  MoveL 3421 to (458.38, 544.47, 60) mm, rotated rx 180 ry 0 rz 160 deg; joints [12.908, 64.671, 4.194, -145.247, 72.379, 168.139]
  Call Extruder(250.39892)
  MoveL 3422 to (457.49, 543.62, 60) mm, rotated rx -180 ry 0 rz 160 deg; joints [12.822, 64.543, 4.5, -145.367, 72.508, 168.272]
  Call Extruder(254.47184)
  MoveL 3423 to (456.59, 542.72, 60) mm, rotated rx -180 ry 0 rz 160 deg; joints [12.729, 64.414, 4.81, -145.496, 72.639, 168.409]
  Set speed (17.7 mm/s)
  Call Extruder(258.50937)
  MoveL 3424 to (455.71, 541.81, 60) mm, rotated rx -180 ry 0 rz 160 deg; joints [12.633, 64.289, 5.114, -145.625, 72.766, 168.543]
  Call Extruder(262.39777)
  MoveL 3425 to (454.88, 540.92, 60) mm, rotated rx 180 ry 0 rz 160 deg; joints [12.537, 64.17, 5.4, -145.753, 72.886, 168.671]
  Set speed (17.7 mm/s)
  Call Extruder(266.46406)
  MoveL 3426 to (454.04, 539.97, 60) mm, rotated rx -180 ry 0 rz 160 deg; joints [12.434, 64.049, 5.695, -145.888, 73.009, 168.804]
  Set speed (17.7 mm/s)
  Call Extruder(270.34791)
  MoveL 3427 to (453.25, 539.04, 60) mm, rotated rx -180 ry 0 rz 160 deg; joints [12.332, 63.935, 5.97, -146.021, 73.124, 168.929]
  Call Extruder(274.31271)
  MoveL 3428 to (452.46, 538.08, 60) mm, rotated rx 180 ry 0 rz 160 deg; joints [12.225, 63.822, 6.246, -146.158, 73.238, 169.056]
  Set speed (17.7 mm/s)
  Call Extruder(278.33345)
  MoveL 3429 to (451.68, 537.1, 60) mm, rotated rx 180 ry 0 rz 160 deg; joints [12.113, 63.71, 6.52, -146.3, 73.352, 169.183]
  Call Extruder(282.32372)
  MoveL 3430 to (450.94, 536.1, 60) mm, rotated rx 180 ry 0 rz 160 deg; joints [11.998, 63.601, 6.786, -146.444, 73.461, 169.307]
  Set speed (17.7 mm/s)
  Call Extruder(286.28959)
  MoveL 3431 to (450.21, 535.09, 60) mm, rotated rx 180 ry 0 rz 160 deg; joints [11.88, 63.495, 7.044, -146.589, 73.567, 169.429]
  Call Extruder(290.26148)
  MoveL 3432 to (449.5, 534.06, 60) mm, rotated rx -180 ry 0 rz 160 deg; joints [11.76, 63.392, 7.297, -146.736, 73.67, 169.55]
  Call Extruder(294.32502)
  MoveL 3433 to (448.81, 533, 60) mm, rotated rx 180 ry 0 rz 160 deg; joints [11.634, 63.29, 7.549, -146.89, 73.772, 169.671]
  Set speed (17.7 mm/s)
  Call Extruder(298.26201)
  MoveL 3434 to (448.15, 531.96, 60) mm, rotated rx 180 ry 0 rz 160 deg; joints [11.508, 63.193, 7.787, -147.041, 73.868, 169.787]
  Set speed (17.7 mm/s)
  Call Extruder(302.15383)
  MoveL 3435 to (447.52, 530.92, 60) mm, rotated rx -180 ry 0 rz 160 deg; joints [11.381, 63.1, 8.016, -147.192, 73.96, 169.9]
  Set speed (17.6 mm/s)
  Call Extruder(306.26935)
  MoveL 3436 to (446.88, 529.8, 60) mm, rotated rx 180 ry 0 rz 160 deg; joints [11.244, 63.005, 8.252, -147.355, 74.054, 170.018]
  Set speed (17.6 mm/s)
  Call Extruder(310.11261)
  MoveL 3437 to (446.3, 528.75, 60) mm, rotated rx 180 ry 0 rz 160 deg; joints [11.113, 62.918, 8.466, -147.508, 74.139, 170.126]
  Set speed (17.7 mm/s)
  Call Extruder(314.10849)
  MoveL 3438 to (445.72, 527.64, 60) mm, rotated rx 180 ry 0 rz 160 deg; joints [10.974, 62.831, 8.682, -147.67, 74.224, 170.237]
  Set speed (17.7 mm/s)
  Call Extruder(318.14964)
  MoveL 3439 to (445.16, 526.51, 60) mm, rotated rx 180 ry 0 rz 160 deg; joints [10.831, 62.746, 8.893, -147.836, 74.307, 170.347]
  Set speed (17.7 mm/s)
  Call Extruder(325.99805)
  MoveL 3440 to (444.13, 524.27, 60) mm, rotated rx 180 ry 0 rz 160 deg; joints [10.544, 62.589, 9.284, -148.164, 74.457, 170.554]
  Set speed (17.6 mm/s)
  Call Extruder(330.16567)
  MoveL 3441 to (443.63, 523.07, 60) mm, rotated rx -180 ry 0 rz 160 deg; joints [10.388, 62.511, 9.478, -148.341, 74.531, 170.661]
  Call Extruder(334.15174)
  MoveL 3442 to (443.17, 521.91, 60) mm, rotated rx -180 ry 0 rz 160 deg; joints [10.236, 62.438, 9.66, -148.512, 74.6, 170.761]
  Set speed (17.7 mm/s)
  Call Extruder(342.11094)
  MoveL 3443 to (442.32, 519.57, 60) mm, rotated rx 180 ry 0 rz 160 deg; joints [9.926, 62.302, 10.001, -148.858, 74.725, 170.955]
  Set speed (17.6 mm/s)
  Call Extruder(346.07808)
  MoveL 3444 to (441.94, 518.39, 60) mm, rotated rx 180 ry 0 rz 160 deg; joints [9.768, 62.24, 10.157, -149.034, 74.781, 171.048]
  Set speed (17.6 mm/s)
  Call Extruder(350.09490)
  MoveL 3445 to (441.57, 517.19, 60) mm, rotated rx 180 ry 0 rz 160 deg; joints [9.606, 62.179, 10.312, -149.212, 74.836, 171.141]
  Set speed (17.6 mm/s)
  Call Extruder(354.07902)
  MoveL 3446 to (441.23, 516, 60) mm, rotated rx -180 ry 0 rz 160 deg; joints [9.443, 62.122, 10.456, -149.391, 74.885, 171.231]
  Set speed (17.6 mm/s)
  Call Extruder(357.89675)
  MoveL 3447 to (440.93, 514.84, 60) mm, rotated rx 180 ry 0 rz 160 deg; joints [9.286, 62.069, 10.589, -149.563, 74.931, 171.315]
  Set speed (17.6 mm/s)
  Call Extruder(362.02810)
  MoveL 3448 to (440.63, 513.59, 60) mm, rotated rx -180 ry 0 rz 160 deg; joints [9.113, 62.016, 10.722, -149.751, 74.974, 171.403]
  Set speed (17.6 mm/s)
  Call Extruder(366.00274)
  MoveL 3449 to (440.36, 512.37, 60) mm, rotated rx -180 ry 0 rz 160 deg; joints [8.945, 61.967, 10.845, -149.933, 75.014, 171.486]
  Set speed (17.7 mm/s)
  Call Extruder(374.01194)
  MoveL 3450 to (439.9, 509.91, 60) mm, rotated rx 180 ry 0 rz 160 deg; joints [8.601, 61.878, 11.069, -150.303, 75.081, 171.647]
  Set speed (17.7 mm/s)
  Call Extruder(381.96597)
  MoveL 3451 to (439.55, 507.44, 60) mm, rotated rx 180 ry 0 rz 160 deg; joints [8.253, 61.803, 11.261, -150.674, 75.131, 171.797]
  Set speed (17.7 mm/s)
  Call Extruder(389.93168)
  MoveL 3452 to (439.29, 504.96, 60) mm, rotated rx 180 ry 0 rz 160 deg; joints [7.9, 61.739, 11.422, -151.049, 75.167, 171.939]
  Set speed (17.7 mm/s)
  Call Extruder(397.72230)
  MoveL 3453 to (439.14, 502.53, 60) mm, rotated rx -180 ry 0 rz 160 deg; joints [7.551, 61.689, 11.55, -151.416, 75.186, 172.069]
  Set speed (17.7 mm/s)
  Call Extruder(405.77297)
  MoveL 3454 to (439.09, 500.01, 60) mm, rotated rx 180 ry 0 rz 160 deg; joints [7.186, 61.649, 11.651, -151.798, 75.19, 172.195]
  Set speed (17.7 mm/s)
  Call Extruder(413.01680)
  MoveL 3455 to (439.13, 497.74, 60) mm, rotated rx 180 ry 0 rz 160 deg; joints [6.856, 61.624, 11.714, -152.141, 75.179, 172.3]
  Set speed (17.7 mm/s)
  Call Extruder(420.09250)
  MoveL 3456 to (439.25, 495.53, 60) mm, rotated rx 180 ry 0 rz 160 deg; joints [6.532, 61.61, 11.75, -152.476, 75.156, 172.396]
  Set speed (17.7 mm/s)
  Call Extruder(427.18898)
  MoveL 3457 to (439.46, 493.32, 60) mm, rotated rx 180 ry 0 rz 160 deg; joints [6.207, 61.606, 11.762, -152.81, 75.119, 172.485]
  Set speed (17.7 mm/s)
  Call Extruder(434.08176)
  MoveL 3458 to (439.73, 491.18, 60) mm, rotated rx 180 ry 0 rz 160 deg; joints [5.891, 61.611, 11.749, -153.133, 75.071, 172.564]
  Call Extruder(441.67457)
  MoveL 3459 to (440.12, 488.84, 60) mm, rotated rx -180 ry 0 rz 160 deg; joints [5.544, 61.627, 11.708, -153.487, 75.004, 172.645]
  Set speed (17.7 mm/s)
  Call Extruder(448.69639)
  MoveL 3460 to (440.56, 486.69, 60) mm, rotated rx 180 ry 0 rz 160 deg; joints [5.224, 61.652, 11.644, -153.811, 74.929, 172.712]
  Call Extruder(455.92149)
  MoveL 3461 to (441.1, 484.49, 60) mm, rotated rx 180 ry 0 rz 160 deg; joints [4.897, 61.687, 11.554, -154.14, 74.838, 172.775]
  Call Extruder(462.99323)
  MoveL 3462 to (441.7, 482.36, 60) mm, rotated rx 180 ry 0 rz 160 deg; joints [4.579, 61.732, 11.44, -154.459, 74.736, 172.83]
  Set speed (17.7 mm/s)
  Call Extruder(470.18160)
  MoveL 3463 to (442.39, 480.22, 60) mm, rotated rx -180 ry 0 rz 160 deg; joints [4.26, 61.788, 11.299, -154.777, 74.619, 172.878]
  Set speed (17.7 mm/s)
  Call Extruder(477.50769)
  MoveL 3464 to (443.18, 478.07, 60) mm, rotated rx 180 ry 0 rz 160 deg; joints [3.939, 61.855, 11.129, -155.096, 74.486, 172.921]
  Set speed (17.7 mm/s)
  Call Extruder(484.67427)
  MoveL 3465 to (444.02, 475.99, 60) mm, rotated rx 180 ry 0 rz 160 deg; joints [3.629, 61.93, 10.939, -155.401, 74.344, 172.957]
  Set speed (17.7 mm/s)
  Call Extruder(491.67065)
  MoveL 3466 to (444.92, 473.99, 60) mm, rotated rx -180 ry 0 rz 160 deg; joints [3.332, 62.013, 10.729, -155.693, 74.192, 172.986]
  Set speed (17.7 mm/s)
  Call Extruder(499.01562)
  MoveL 3467 to (445.94, 471.93, 60) mm, rotated rx -180 ry 0 rz 160 deg; joints [3.026, 62.111, 10.483, -155.992, 74.019, 173.009]
  Set speed (17.6 mm/s)
  Call Extruder(506.01239)
  MoveL 3468 to (446.99, 470.01, 60) mm, rotated rx 180 ry 0 rz 160 deg; joints [2.74, 62.212, 10.227, -156.269, 73.844, 173.026]
  Set speed (17.7 mm/s)
  Call Extruder(513.18194)
  MoveL 3469 to (448.13, 468.08, 60) mm, rotated rx -180 ry 0 rz 160 deg; joints [2.455, 62.326, 9.941, -156.544, 73.651, 173.037]
  Set speed (17.7 mm/s)
  Call Extruder(520.42302)
  MoveL 3470 to (449.35, 466.17, 60) mm, rotated rx -180 ry 0 rz 160 deg; joints [2.173, 62.451, 9.628, -156.813, 73.445, 173.042]
  Set speed (17.7 mm/s)
  Call Extruder(527.57955)
  MoveL 3471 to (450.62, 464.33, 60) mm, rotated rx -180 ry 0 rz 160 deg; joints [1.903, 62.584, 9.296, -157.07, 73.229, 173.041]
  Set speed (17.7 mm/s)
  Call Extruder(534.77776)
  MoveL 3472 to (451.98, 462.53, 60) mm, rotated rx -180 ry 0 rz 160 deg; joints [1.64, 62.727, 8.94, -157.318, 73, 173.033]
  Call Extruder(541.94995)
  MoveL 3473 to (453.39, 460.79, 60) mm, rotated rx 180 ry 0 rz 160 deg; joints [1.386, 62.88, 8.562, -157.555, 72.761, 173.02]
  Set speed (17.7 mm/s)
  Call Extruder(549.06578)
  MoveL 3474 to (454.86, 459.11, 60) mm, rotated rx 180 ry 0 rz 160 deg; joints [1.143, 63.039, 8.166, -157.779, 72.513, 173.002]
  Set speed (17.7 mm/s)
  Call Extruder(556.16490)
  MoveL 3475 to (456.38, 457.49, 60) mm, rotated rx 180 ry 0 rz 160 deg; joints [0.91, 63.208, 7.75, -157.993, 72.256, 172.978]
  Set speed (17.7 mm/s)
  Call Extruder(563.37874)
  MoveL 3476 to (457.99, 455.9, 60) mm, rotated rx -180 ry 0 rz 160 deg; joints [0.683, 63.388, 7.308, -158.198, 71.984, 172.947]
  Set speed (17.7 mm/s)
  Call Extruder(570.70409)
  MoveL 3477 to (459.68, 454.35, 60) mm, rotated rx 180 ry 0 rz 160 deg; joints [0.463, 63.58, 6.837, -158.394, 71.698, 172.91]
  Set speed (17.7 mm/s)
  Call Extruder(577.80064)
  MoveL 3478 to (461.37, 452.91, 60) mm, rotated rx 180 ry 0 rz 160 deg; joints [0.26, 63.774, 6.362, -158.571, 71.412, 172.869]
  Set speed (17.7 mm/s)
  Call Extruder(584.88132)
  MoveL 3479 to (463.11, 451.53, 60) mm, rotated rx 180 ry 0 rz 160 deg; joints [0.068, 63.977, 5.87, -158.737, 71.118, 172.822]
  Set speed (17.7 mm/s)
  Call Extruder(592.12824)
  MoveL 3480 to (464.94, 450.19, 60) mm, rotated rx -180 ry 0 rz 160 deg; joints [-0.118, 64.192, 5.348, -158.893, 70.809, 172.769]
  Set speed (17.7 mm/s)
  Call Extruder(599.20393)
  MoveL 3481 to (466.77, 448.95, 60) mm, rotated rx -180 ry 0 rz 160 deg; joints [-0.288, 64.41, 4.82, -159.034, 70.499, 172.71]
  Set speed (17.7 mm/s)
  Call Extruder(606.45847)
  MoveL 3482 to (468.7, 447.75, 60) mm, rotated rx 180 ry 0 rz 160 deg; joints [-0.452, 64.642, 4.262, -159.164, 70.173, 172.645]
  Set speed (17.7 mm/s)
  Call Extruder(613.61813)
  MoveL 3483 to (470.64, 446.63, 60) mm, rotated rx 180 ry 0 rz 160 deg; joints [-0.602, 64.879, 3.695, -159.28, 69.845, 172.574]
  Set speed (17.7 mm/s)
  Call Extruder(620.78178)
  MoveL 3484 to (472.62, 445.59, 60) mm, rotated rx 180 ry 0 rz 160 deg; joints [-0.741, 65.123, 3.112, -159.383, 69.509, 172.498]
  Set speed (17.7 mm/s)
  Call Extruder(627.85751)
  MoveL 3485 to (474.62, 444.63, 60) mm, rotated rx -180 ry 0 rz 160 deg; joints [-0.867, 65.372, 2.52, -159.471, 69.172, 172.416]
  Call Extruder(635.11103)
  MoveL 3486 to (476.7, 443.72, 60) mm, rotated rx -180 ry 0 rz 160 deg; joints [-0.985, 65.633, 1.9, -159.548, 68.82, 172.326]
  Set speed (17.7 mm/s)
  Call Extruder(642.12717)
  MoveL 3487 to (478.75, 442.92, 60) mm, rotated rx -180 ry 0 rz 160 deg; joints [-1.087, 65.894, 1.286, -159.609, 68.475, 172.233]
  Set speed (17.7 mm/s)
  Call Extruder(649.44940)
  MoveL 3488 to (480.91, 442.16, 60) mm, rotated rx 180 ry 0 rz 160 deg; joints [-1.183, 66.172, 0.632, -159.659, 68.109, 172.13]
  Set speed (17.7 mm/s)
  Call Extruder(656.54664)
  MoveL 3489 to (483.03, 441.5, 60) mm, rotated rx 180 ry 0 rz 160 deg; joints [-1.264, 66.447, -0.015, -159.694, 67.751, 172.024]
  Set speed (17.7 mm/s)
  Call Extruder(663.55363)
  MoveL 3490 to (485.15, 440.93, 60) mm, rotated rx -180 ry 0 rz 160 deg; joints [-1.334, 66.726, -0.664, -159.715, 67.393, 171.913]
  Call Extruder(670.92630)
  MoveL 3491 to (487.39, 440.41, 60) mm, rotated rx -180 ry 0 rz 160 deg; joints [-1.395, 67.024, -1.359, -159.723, 67.013, 171.79]
  Set speed (17.7 mm/s)
  Call Extruder(677.95259)
  MoveL 3492 to (489.55, 439.99, 60) mm, rotated rx -180 ry 0 rz 160 deg; joints [-1.442, 67.315, -2.031, -159.717, 66.647, 171.666]
  Call Extruder(684.84672)
  MoveL 3493 to (491.69, 439.66, 60) mm, rotated rx 180 ry 0 rz 160 deg; joints [-1.479, 67.604, -2.699, -159.699, 66.287, 171.538]
  Call Extruder(692.33816)
  MoveL 3494 to (494.01, 439.38, 60) mm, rotated rx -180 ry 0 rz 160 deg; joints [-1.506, 67.924, -3.435, -159.665, 65.893, 171.392]
  Set speed (17.7 mm/s)
  Call Extruder(699.51358)
  MoveL 3495 to (496.25, 439.21, 60) mm, rotated rx 180 ry 0 rz 160 deg; joints [-1.522, 68.236, -4.148, -159.619, 65.514, 171.246]
  Call Extruder(706.76277)
  MoveL 3496 to (498.52, 439.11, 60) mm, rotated rx 180 ry 0 rz 160 deg; joints [-1.527, 68.554, -4.876, -159.559, 65.13, 171.091]
  Call Extruder(713.85821)
  MoveL 3497 to (500.74, 439.1, 60) mm, rotated rx -180 ry 0 rz 160 deg; joints [-1.521, 68.871, -5.595, -159.486, 64.754, 170.933]
  Set speed (17.7 mm/s)
  Call Extruder(720.88825)
  MoveL 3498 to (502.94, 439.16, 60) mm, rotated rx 180 ry 0 rz 160 deg; joints [-1.505, 69.187, -6.313, -159.402, 64.381, 170.77]
  Call Extruder(728.18043)
  MoveL 3499 to (505.22, 439.31, 60) mm, rotated rx 180 ry 0 rz 160 deg; joints [-1.478, 69.52, -7.063, -159.301, 63.994, 170.593]
  Set speed (17.7 mm/s)
  Call Extruder(735.41102)
  MoveL 3500 to (507.47, 439.55, 60) mm, rotated rx 180 ry 0 rz 160 deg; joints [-1.441, 69.852, -7.81, -159.188, 63.612, 170.411]
  Set speed (17.7 mm/s)
  Call Extruder(742.49479)
  MoveL 3501 to (509.66, 439.86, 60) mm, rotated rx 180 ry 0 rz 160 deg; joints [-1.396, 70.18, -8.545, -159.065, 63.239, 170.227]
  Set speed (17.6 mm/s)
  Call Extruder(749.70308)
  MoveL 3502 to (511.88, 440.26, 60) mm, rotated rx -180 ry 0 rz 160 deg; joints [-1.339, 70.515, -9.296, -158.928, 62.862, 170.032]
  Set speed (17.7 mm/s)
  Call Extruder(756.88945)
  MoveL 3503 to (514.08, 440.74, 60) mm, rotated rx -180 ry 0 rz 160 deg; joints [-1.274, 70.852, -10.045, -158.778, 62.488, 169.83]
  Set speed (17.7 mm/s)
  Call Extruder(763.93252)
  MoveL 3504 to (516.21, 441.29, 60) mm, rotated rx 180 ry 0 rz 160 deg; joints [-1.201, 71.183, -10.781, -158.619, 62.124, 169.627]
  Set speed (17.7 mm/s)
  Call Extruder(771.15493)
  MoveL 3505 to (518.38, 441.93, 60) mm, rotated rx 180 ry 0 rz 160 deg; joints [-1.116, 71.524, -11.536, -158.445, 61.754, 169.411]
  Call Extruder(778.20140)
  MoveL 3506 to (520.47, 442.63, 60) mm, rotated rx -180 ry 0 rz 160 deg; joints [-1.026, 71.857, -12.271, -158.263, 61.398, 169.194]
  Set speed (17.7 mm/s)
  Call Extruder(785.48617)
  MoveL 3507 to (522.61, 443.44, 60) mm, rotated rx -180 ry 0 rz 160 deg; joints [-0.923, 72.202, -13.029, -158.064, 61.033, 168.964]
  Set speed (17.7 mm/s)
  Call Extruder(792.88462)
  MoveL 3508 to (524.74, 444.34, 60) mm, rotated rx 180 ry 0 rz 160 deg; joints [-0.81, 72.551, -13.795, -157.85, 60.669, 168.722]
  Set speed (17.7 mm/s)
  Call Extruder(799.85949)
  MoveL 3509 to (526.72, 445.26, 60) mm, rotated rx 180 ry 0 rz 160 deg; joints [-0.696, 72.88, -14.515, -157.637, 60.33, 168.489]
  Set speed (17.7 mm/s)
  Call Extruder(807.02755)
  MoveL 3510 to (528.71, 446.28, 60) mm, rotated rx 180 ry 0 rz 160 deg; joints [-0.57, 73.217, -15.249, -157.409, 59.988, 168.244]
  Set speed (17.7 mm/s)
  Call Extruder(814.23835)
  MoveL 3511 to (530.68, 447.38, 60) mm, rotated rx 180 ry 0 rz 160 deg; joints [-0.437, 73.554, -15.981, -157.169, 59.65, 167.991]
  Set speed (17.7 mm/s)
  Call Extruder(821.30859)
  MoveL 3512 to (532.58, 448.53, 60) mm, rotated rx -180 ry 0 rz 160 deg; joints [-0.299, 73.882, -16.693, -156.924, 59.326, 167.738]
  Call Extruder(828.55700)
  MoveL 3513 to (534.47, 449.78, 60) mm, rotated rx -180 ry 0 rz 160 deg; joints [-0.149, 74.215, -17.414, -156.663, 59.002, 167.473]
  Call Extruder(835.64231)
  MoveL 3514 to (536.27, 451.07, 60) mm, rotated rx 180 ry 0 rz 160 deg; joints [0.003, 74.538, -18.111, -156.399, 58.693, 167.209]
  Set speed (17.7 mm/s)
  Call Extruder(842.84270)
  MoveL 3515 to (538.06, 452.45, 60) mm, rotated rx 180 ry 0 rz 160 deg; joints [0.165, 74.863, -18.81, -156.122, 58.386, 166.936]
  Set speed (17.7 mm/s)
  Call Extruder(850.00063)
  MoveL 3516 to (539.78, 453.88, 60) mm, rotated rx 180 ry 0 rz 160 deg; joints [0.332, 75.181, -19.492, -155.838, 58.091, 166.66]
  Set speed (17.7 mm/s)
  Call Extruder(857.35471)
  MoveL 3517 to (541.5, 455.41, 60) mm, rotated rx -180 ry 0 rz 160 deg; joints [0.51, 75.503, -20.181, -155.539, 57.798, 166.373]
  Set speed (17.7 mm/s)
  Call Extruder(864.32574)
  MoveL 3518 to (543.07, 456.93, 60) mm, rotated rx -180 ry 0 rz 160 deg; joints [0.685, 75.803, -20.823, -155.249, 57.529, 166.098]
  Set speed (17.7 mm/s)
  Call Extruder(868.29280)
  MoveL 3519 to (543.94, 457.82, 60) mm, rotated rx -180 ry 0 rz 160 deg; joints [0.787, 75.97, -21.18, -155.08, 57.382, 165.94]
  Set speed (17.7 mm/s)
  Call Extruder(872.16707)
  MoveL 3520 to (544.77, 458.7, 60) mm, rotated rx 180 ry 0 rz 160 deg; joints [0.888, 76.133, -21.526, -154.914, 57.24, 165.785]
  Set speed (17.7 mm/s)
  Call Extruder(876.17456)
  MoveL 3521 to (545.61, 459.63, 60) mm, rotated rx -180 ry 0 rz 160 deg; joints [0.994, 76.298, -21.879, -154.74, 57.097, 165.624]
  Call Extruder(880.12274)
  MoveL 3522 to (546.42, 460.56, 60) mm, rotated rx -180 ry 0 rz 160 deg; joints [1.1, 76.46, -22.222, -154.567, 56.959, 165.464]
  Set speed (17.7 mm/s)
  Call Extruder(884.11982)
  MoveL 3523 to (547.22, 461.52, 60) mm, rotated rx -180 ry 0 rz 160 deg; joints [1.209, 76.621, -22.564, -154.39, 56.823, 165.302]
  Set speed (17.7 mm/s)
  Call Extruder(888.15091)
  MoveL 3524 to (548.01, 462.51, 60) mm, rotated rx 180 ry 0 rz 160 deg; joints [1.321, 76.78, -22.903, -154.21, 56.69, 165.139]
  Set speed (17.7 mm/s)
  Call Extruder(892.09605)
  MoveL 3525 to (548.76, 463.49, 60) mm, rotated rx 180 ry 0 rz 160 deg; joints [1.432, 76.934, -23.228, -154.033, 56.564, 164.978]
  Set speed (17.7 mm/s)
  Call Extruder(896.05523)
  MoveL 3526 to (549.49, 464.49, 60) mm, rotated rx -180 ry 0 rz 160 deg; joints [1.545, 77.086, -23.55, -153.853, 56.441, 164.817]
  Call Extruder(900.07180)
  MoveL 3527 to (550.21, 465.52, 60) mm, rotated rx -180 ry 0 rz 160 deg; joints [1.66, 77.237, -23.87, -153.669, 56.32, 164.653]
  Set speed (17.6 mm/s)
  Call Extruder(904.02046)
  MoveL 3528 to (550.9, 466.55, 60) mm, rotated rx -180 ry 0 rz 160 deg; joints [1.775, 77.383, -24.179, -153.488, 56.205, 164.492]
  Set speed (17.7 mm/s)
  Call Extruder(908.03453)
  MoveL 3529 to (551.58, 467.6, 60) mm, rotated rx 180 ry 0 rz 160 deg; joints [1.894, 77.529, -24.487, -153.302, 56.092, 164.328]
  Call Extruder(912.01280)
  MoveL 3530 to (552.23, 468.66, 60) mm, rotated rx -180 ry 0 rz 160 deg; joints [2.012, 77.67, -24.785, -153.116, 55.984, 164.166]
  Set speed (17.7 mm/s)
  Call Extruder(916.05485)
  MoveL 3531 to (552.87, 469.75, 60) mm, rotated rx 180 ry 0 rz 160 deg; joints [2.134, 77.811, -25.081, -152.927, 55.879, 164.002]
  Set speed (17.6 mm/s)
  Call Extruder(921.15306)
  MoveL 3532 to (553.65, 471.15, 60) mm, rotated rx -180 ry 0 rz 160 deg; joints [2.289, 77.983, -25.444, -152.688, 55.753, 163.795]
  Call Extruder(923.98862)
  MoveL 3533 to (554.06, 471.93, 60) mm, rotated rx 180 ry 0 rz 160 deg; joints [2.376, 78.076, -25.639, -152.554, 55.686, 163.681]
  Set speed (17.7 mm/s)
  Call Extruder(927.92565)
  MoveL 3534 to (554.61, 473.03, 60) mm, rotated rx 180 ry 0 rz 160 deg; joints [2.498, 78.204, -25.907, -152.368, 55.596, 163.523]
  Set speed (17.7 mm/s)
  Call Extruder(931.94237)
  MoveL 3535 to (555.16, 474.16, 60) mm, rotated rx 180 ry 0 rz 160 deg; joints [2.624, 78.33, -26.171, -152.178, 55.509, 163.362]
  Set speed (17.7 mm/s)
  Call Extruder(935.87944)
  MoveL 3536 to (555.67, 475.28, 60) mm, rotated rx -180 ry 0 rz 160 deg; joints [2.748, 78.45, -26.424, -151.991, 55.428, 163.205]
  Set speed (17.6 mm/s)
  Call Extruder(943.97320)
  MoveL 3537 to (556.65, 477.62, 60) mm, rotated rx -180 ry 0 rz 160 deg; joints [3.007, 78.685, -26.916, -151.606, 55.277, 162.886]
  Set speed (17.6 mm/s)
  Call Extruder(947.91335)
  MoveL 3538 to (557.08, 478.77, 60) mm, rotated rx 180 ry 0 rz 160 deg; joints [3.134, 78.792, -27.141, -151.419, 55.211, 162.733]
  Set speed (17.6 mm/s)
  Call Extruder(951.77830)
  MoveL 3539 to (557.5, 479.9, 60) mm, rotated rx -180 ry 0 rz 160 deg; joints [3.259, 78.896, -27.358, -151.236, 55.149, 162.584]
  Call Extruder(955.89683)
  MoveL 3540 to (557.91, 481.12, 60) mm, rotated rx -180 ry 0 rz 160 deg; joints [3.394, 79.001, -27.577, -151.041, 55.09, 162.427]
  Set speed (17.6 mm/s)
  Call Extruder(959.91891)
  MoveL 3541 to (558.29, 482.32, 60) mm, rotated rx 180 ry 0 rz 160 deg; joints [3.526, 79.101, -27.786, -150.85, 55.034, 162.275]
  Set speed (17.7 mm/s)
  Call Extruder(967.71701)
  MoveL 3542 to (558.95, 484.67, 60) mm, rotated rx 180 ry 0 rz 160 deg; joints [3.785, 79.28, -28.16, -150.482, 54.944, 161.985]
  Set speed (17.6 mm/s)
  Call Extruder(971.84165)
  MoveL 3543 to (559.26, 485.92, 60) mm, rotated rx -180 ry 0 rz 160 deg; joints [3.924, 79.366, -28.34, -150.289, 54.905, 161.836]
  Call Extruder(975.71381)
  MoveL 3544 to (559.53, 487.1, 60) mm, rotated rx 180 ry 0 rz 160 deg; joints [4.054, 79.446, -28.506, -150.108, 54.871, 161.697]
  Set speed (17.7 mm/s)
  Call Extruder(983.59562)
  MoveL 3545 to (560, 489.52, 60) mm, rotated rx 180 ry 0 rz 160 deg; joints [4.321, 79.591, -28.808, -149.742, 54.82, 161.422]
  Set speed (17.7 mm/s)
  Call Extruder(991.63549)
  MoveL 3546 to (560.38, 492.01, 60) mm, rotated rx -180 ry 0 rz 160 deg; joints [4.596, 79.721, -29.079, -149.374, 54.787, 161.152]
  Set speed (17.7 mm/s)
  Call Extruder(999.76645)
  MoveL 3547 to (560.67, 494.54, 60) mm, rotated rx -180 ry 0 rz 160 deg; joints [4.875, 79.832, -29.31, -149.006, 54.774, 160.889]
  Call Extruder(1007.63307)
  MoveL 3548 to (560.84, 497, 60) mm, rotated rx -180 ry 0 rz 160 deg; joints [5.148, 79.92, -29.493, -148.657, 54.783, 160.648]
  Set speed (17.7 mm/s)
  Call Extruder(1015.58635)
  MoveL 3549 to (560.91, 499.49, 60) mm, rotated rx -180 ry 0 rz 160 deg; joints [5.424, 79.989, -29.637, -148.311, 54.811, 160.416]
  Set speed (17.7 mm/s)
  Call Extruder(1023.42990)
  MoveL 3550 to (560.88, 501.94, 60) mm, rotated rx 180 ry 0 rz 160 deg; joints [5.698, 80.037, -29.736, -147.977, 54.859, 160.201]
  Set speed (17.7 mm/s)
  Call Extruder(1031.49963)
  MoveL 3551 to (560.75, 504.46, 60) mm, rotated rx 180 ry 0 rz 160 deg; joints [5.98, 80.066, -29.796, -147.641, 54.929, 159.995]
  Call Extruder(1039.46843)
  MoveL 3552 to (560.51, 506.95, 60) mm, rotated rx 180 ry 0 rz 160 deg; joints [6.258, 80.073, -29.812, -147.318, 55.018, 159.806]
  Call Extruder(1047.51753)
  MoveL 3553 to (560.17, 509.45, 60) mm, rotated rx -180 ry 0 rz 160 deg; joints [6.54, 80.059, -29.783, -147.002, 55.128, 159.632]
  Set speed (17.7 mm/s)
  Call Extruder(1055.37383)
  MoveL 3554 to (559.74, 511.87, 60) mm, rotated rx 180 ry 0 rz 160 deg; joints [6.814, 80.026, -29.714, -146.702, 55.254, 159.477]
  Call Extruder(1063.39954)
  MoveL 3555 to (559.2, 514.32, 60) mm, rotated rx 180 ry 0 rz 160 deg; joints [7.094, 79.971, -29.6, -146.407, 55.402, 159.335]
  Set speed (17.7 mm/s)
  Call Extruder(1071.21656)
  MoveL 3556 to (558.58, 516.69, 60) mm, rotated rx -180 ry 0 rz 160 deg; joints [7.365, 79.898, -29.447, -146.129, 55.564, 159.214]
  Set speed (17.6 mm/s)
  Call Extruder(1075.37612)
  MoveL 3557 to (558.21, 517.93, 60) mm, rotated rx -180 ry 0 rz 160 deg; joints [7.508, 79.85, -29.347, -145.986, 55.658, 159.158]
  Set speed (17.6 mm/s)
  Call Extruder(1079.17724)
  MoveL 3558 to (557.85, 519.07, 60) mm, rotated rx -180 ry 0 rz 160 deg; joints [7.64, 79.804, -29.251, -145.857, 55.746, 159.108]
  Set speed (17.7 mm/s)
  Call Extruder(1087.36494)
  MoveL 3559 to (557, 521.48, 60) mm, rotated rx 180 ry 0 rz 160 deg; joints [7.921, 79.686, -29.006, -145.588, 55.951, 159.016]
  Set speed (17.7 mm/s)
  Call Extruder(1095.08205)
  MoveL 3560 to (556.1, 523.72, 60) mm, rotated rx 180 ry 0 rz 160 deg; joints [8.184, 79.556, -28.736, -145.346, 56.161, 158.947]
  Set speed (17.6 mm/s)
  Call Extruder(1099.19827)
  MoveL 3561 to (555.58, 524.9, 60) mm, rotated rx -180 ry 0 rz 160 deg; joints [8.323, 79.479, -28.575, -145.222, 56.28, 158.918]
  Set speed (17.6 mm/s)
  Call Extruder(1102.99136)
  MoveL 3562 to (555.09, 525.98, 60) mm, rotated rx 180 ry 0 rz 160 deg; joints [8.451, 79.405, -28.422, -145.108, 56.392, 158.893]
  Set speed (17.6 mm/s)
  Call Extruder(1105.96710)
  MoveL 3563 to (554.69, 526.82, 60) mm, rotated rx 180 ry 0 rz 160 deg; joints [8.551, 79.345, -28.296, -145.021, 56.482, 158.876]
  Set speed (17.6 mm/s)
  Call Extruder(1111.16558)
  MoveL 3564 to (553.96, 528.27, 60) mm, rotated rx -180 ry 0 rz 160 deg; joints [8.725, 79.232, -28.06, -144.874, 56.645, 158.854]
  Set speed (17.7 mm/s)
  Call Extruder(1115.08771)
  MoveL 3565 to (553.37, 529.35, 60) mm, rotated rx -180 ry 0 rz 160 deg; joints [8.855, 79.141, -27.87, -144.766, 56.772, 158.842]
  Set speed (17.6 mm/s)
  Call Extruder(1119.14376)
  MoveL 3566 to (552.75, 530.46, 60) mm, rotated rx 180 ry 0 rz 160 deg; joints [8.989, 79.043, -27.665, -144.657, 56.908, 158.834]
  Set speed (17.7 mm/s)
  Call Extruder(1122.98241)
  MoveL 3567 to (552.14, 531.49, 60) mm, rotated rx 180 ry 0 rz 160 deg; joints [9.115, 78.947, -27.464, -144.556, 57.039, 158.83]
  Set speed (17.7 mm/s)
  Call Extruder(1126.41961)
  MoveL 3568 to (551.57, 532.41, 60) mm, rotated rx 180 ry 0 rz 160 deg; joints [9.227, 78.857, -27.277, -144.469, 57.159, 158.83]
  Set speed (17.7 mm/s)
  Call Extruder(1131.07197)
  MoveL 3569 to (550.79, 533.63, 60) mm, rotated rx 180 ry 0 rz 160 deg; joints [9.378, 78.731, -27.013, -144.353, 57.326, 158.835]
  Set speed (17.7 mm/s)
  Call Extruder(1135.03970)
  MoveL 3570 to (550.09, 534.66, 60) mm, rotated rx -180 ry 0 rz 160 deg; joints [9.505, 78.619, -26.778, -144.258, 57.472, 158.844]
  Call Extruder(1138.93510)
  MoveL 3571 to (549.39, 535.65, 60) mm, rotated rx -180 ry 0 rz 160 deg; joints [9.63, 78.506, -26.54, -144.166, 57.617, 158.856]
  Call Extruder(1142.95939)
  MoveL 3572 to (548.64, 536.67, 60) mm, rotated rx 180 ry 0 rz 160 deg; joints [9.757, 78.385, -26.287, -144.075, 57.771, 158.873]
  Set speed (17.7 mm/s)
  Call Extruder(1146.90899)
  MoveL 3573 to (547.88, 537.65, 60) mm, rotated rx -180 ry 0 rz 160 deg; joints [9.881, 78.262, -26.03, -143.988, 57.925, 158.894]
  Set speed (17.7 mm/s)
  Call Extruder(1150.87614)
  MoveL 3574 to (547.11, 538.62, 60) mm, rotated rx 180 ry 0 rz 160 deg; joints [10.005, 78.136, -25.764, -143.903, 58.082, 158.918]
  Set speed (17.7 mm/s)
  Call Extruder(1154.87895)
  MoveL 3575 to (546.3, 539.57, 60) mm, rotated rx 180 ry 0 rz 160 deg; joints [10.129, 78.004, -25.488, -143.82, 58.243, 158.947]
  Set speed (17.7 mm/s)
  Call Extruder(1158.89048)
  MoveL 3576 to (545.48, 540.52, 60) mm, rotated rx 180 ry 0 rz 160 deg; joints [10.251, 77.87, -25.204, -143.74, 58.407, 158.98]
  Set speed (17.7 mm/s)
  Call Extruder(1162.94185)
  MoveL 3577 to (544.62, 541.46, 60) mm, rotated rx -180 ry 0 rz 160 deg; joints [10.374, 77.731, -24.911, -143.661, 58.575, 159.016]
  Set speed (17.6 mm/s)
  Call Extruder(1166.20153)
  MoveL 3578 to (543.92, 542.2, 60) mm, rotated rx -180 ry 0 rz 160 deg; joints [10.472, 77.616, -24.67, -143.6, 58.712, 159.049]
  Call Extruder(1170.78283)
  MoveL 3579 to (542.92, 543.22, 60) mm, rotated rx 180 ry 0 rz 160 deg; joints [10.607, 77.452, -24.324, -143.518, 58.907, 159.099]
  Set speed (17.7 mm/s)
  Call Extruder(1174.82308)
  MoveL 3580 to (542.01, 544.1, 60) mm, rotated rx -180 ry 0 rz 160 deg; joints [10.726, 77.304, -24.01, -143.448, 59.082, 159.147]
  Set speed (17.7 mm/s)
  Call Extruder(1178.74465)
  MoveL 3581 to (541.11, 544.94, 60) mm, rotated rx -180 ry 0 rz 160 deg; joints [10.839, 77.157, -23.7, -143.382, 59.253, 159.197]
  Call Extruder(1182.78523)
  MoveL 3582 to (540.17, 545.78, 60) mm, rotated rx 180 ry 0 rz 160 deg; joints [10.955, 77.003, -23.375, -143.317, 59.432, 159.252]
  Set speed (17.7 mm/s)
  Call Extruder(1186.72339)
  MoveL 3583 to (539.24, 546.59, 60) mm, rotated rx 180 ry 0 rz 160 deg; joints [11.066, 76.851, -23.052, -143.257, 59.608, 159.309]
  Set speed (17.7 mm/s)
  Call Extruder(1190.68443)
  MoveL 3584 to (538.28, 547.38, 60) mm, rotated rx -180 ry 0 rz 160 deg; joints [11.177, 76.695, -22.722, -143.198, 59.787, 159.369]
  Set speed (17.6 mm/s)
  Call Extruder(1194.72892)
  MoveL 3585 to (537.29, 548.16, 60) mm, rotated rx 180 ry 0 rz 160 deg; joints [11.288, 76.534, -22.379, -143.141, 59.971, 159.435]
  Set speed (17.6 mm/s)
  Call Extruder(1198.65969)
  MoveL 3586 to (536.31, 548.9, 60) mm, rotated rx 180 ry 0 rz 160 deg; joints [11.394, 76.374, -22.04, -143.088, 60.152, 159.502]
  Set speed (17.7 mm/s)
  Call Extruder(1202.66778)
  MoveL 3587 to (535.3, 549.64, 60) mm, rotated rx -180 ry 0 rz 160 deg; joints [11.501, 76.21, -21.69, -143.036, 60.338, 159.573]
  Set speed (17.7 mm/s)
  Call Extruder(1206.66997)
  MoveL 3588 to (534.27, 550.36, 60) mm, rotated rx -180 ry 0 rz 160 deg; joints [11.606, 76.043, -21.335, -142.987, 60.525, 159.647]
  Call Extruder(1210.71298)
  MoveL 3589 to (533.21, 551.06, 60) mm, rotated rx -180 ry 0 rz 160 deg; joints [11.711, 75.872, -20.971, -142.94, 60.715, 159.726]
  Set speed (17.7 mm/s)
  Call Extruder(1214.67331)
  MoveL 3590 to (532.17, 551.72, 60) mm, rotated rx 180 ry 0 rz 160 deg; joints [11.811, 75.704, -20.611, -142.896, 60.903, 159.805]
  Set speed (17.6 mm/s)
  Call Extruder(1218.61209)
  MoveL 3591 to (531.12, 552.36, 60) mm, rotated rx -180 ry 0 rz 160 deg; joints [11.91, 75.534, -20.248, -142.856, 61.091, 159.887]
  Set speed (17.6 mm/s)
  Call Extruder(1222.58771)
  MoveL 3592 to (530.04, 552.99, 60) mm, rotated rx -180 ry 0 rz 160 deg; joints [12.007, 75.361, -19.879, -142.817, 61.281, 159.973]
  Set speed (17.7 mm/s)
  Call Extruder(1226.49865)
  MoveL 3593 to (528.97, 553.58, 60) mm, rotated rx 180 ry 0 rz 160 deg; joints [12.101, 75.19, -19.511, -142.781, 61.469, 160.06]
  Set speed (17.7 mm/s)
  Call Extruder(1232.61058)
  MoveL 3594 to (527.27, 554.47, 60) mm, rotated rx 180 ry 0 rz 160 deg; joints [12.245, 74.918, -18.929, -142.729, 61.766, 160.2]
  Set speed (17.7 mm/s)
  Call Extruder(1238.37297)
  MoveL 3595 to (525.64, 555.25, 60) mm, rotated rx -180 ry 0 rz 160 deg; joints [12.376, 74.659, -18.371, -142.686, 62.047, 160.34]
  Set speed (17.6 mm/s)
  Call Extruder(1246.39416)
  MoveL 3596 to (523.35, 556.26, 60) mm, rotated rx 180 ry 0 rz 160 deg; joints [12.55, 74.295, -17.586, -142.634, 62.44, 160.541]
  Set speed (17.6 mm/s)
  Call Extruder(1250.48223)
  MoveL 3597 to (522.16, 556.73, 60) mm, rotated rx -180 ry 0 rz 160 deg; joints [12.636, 74.108, -17.181, -142.612, 62.642, 160.648]
  Set speed (17.6 mm/s)
  Call Extruder(1254.26738)
  MoveL 3598 to (521.06, 557.16, 60) mm, rotated rx 180 ry 0 rz 160 deg; joints [12.714, 73.934, -16.805, -142.592, 62.828, 160.749]
  Set speed (17.7 mm/s)
  Call Extruder(1262.39115)
  MoveL 3599 to (518.65, 557.98, 60) mm, rotated rx -180 ry 0 rz 160 deg; joints [12.873, 73.557, -15.988, -142.559, 63.23, 160.972]
  Set speed (17.6 mm/s)
  Call Extruder(1266.41086)
  MoveL 3600 to (517.45, 558.35, 60) mm, rotated rx 180 ry 0 rz 160 deg; joints [12.948, 73.369, -15.58, -142.547, 63.429, 161.086]
  Call Extruder(1270.27929)
  MoveL 3601 to (516.29, 558.69, 60) mm, rotated rx 180 ry 0 rz 160 deg; joints [13.019, 73.189, -15.187, -142.537, 63.621, 161.197]
  Set speed (17.6 mm/s)
  Call Extruder(1273.85715)
  MoveL 3602 to (515.21, 558.98, 60) mm, rotated rx 180 ry 0 rz 160 deg; joints [13.082, 73.021, -14.821, -142.53, 63.798, 161.302]
  Set speed (17.6 mm/s)
  Call Extruder(1278.26443)
  MoveL 3603 to (513.87, 559.31, 60) mm, rotated rx -180 ry 0 rz 160 deg; joints [13.157, 72.814, -14.37, -142.523, 64.016, 161.433]
  Set speed (17.7 mm/s)
  Call Extruder(1286.33939)
  MoveL 3604 to (511.4, 559.84, 60) mm, rotated rx -180 ry 0 rz 160 deg; joints [13.287, 72.434, -13.537, -142.519, 64.416, 161.679]
  Set speed (17.6 mm/s)
  Call Extruder(1294.36497)
  MoveL 3605 to (508.93, 560.25, 60) mm, rotated rx -180 ry 0 rz 160 deg; joints [13.406, 72.054, -12.704, -142.525, 64.813, 161.931]
  Set speed (17.6 mm/s)
  Call Extruder(1302.16248)
  MoveL 3606 to (506.51, 560.56, 60) mm, rotated rx 180 ry 0 rz 160 deg; joints [13.511, 71.686, -11.893, -142.541, 65.197, 162.182]
  Set speed (17.6 mm/s)
  Call Extruder(1310.25608)
  MoveL 3607 to (503.99, 560.78, 60) mm, rotated rx 180 ry 0 rz 160 deg; joints [13.61, 71.304, -11.048, -142.566, 65.594, 162.448]
  Set speed (17.7 mm/s)
  Call Extruder(1318.28261)
  MoveL 3608 to (501.48, 560.89, 60) mm, rotated rx 180 ry 0 rz 160 deg; joints [13.696, 70.926, -10.21, -142.602, 65.986, 162.718]
  Set speed (17.7 mm/s)
  Call Extruder(1326.14950)
  MoveL 3609 to (499.01, 560.9, 60) mm, rotated rx 180 ry 0 rz 160 deg; joints [13.77, 70.557, -9.389, -142.646, 66.367, 162.987]
  Set speed (10.0 mm/s)
  MoveL 3610 to (499.01, 560.9, 64) mm, rotated rx -180 ry 0 rz 160 deg; joints [13.77, 69.876, -8.978, -142.574, 66.152, 162.807]
  Set speed (120.0 mm/s)
  MoveL 3611 to (499, 561.68, 64) mm, rotated rx -180 ry 0 rz 160 deg; joints [13.863, 69.902, -9.036, -142.467, 66.155, 162.746]
  Set speed (17.7 mm/s)
  Call Extruder(1334.25845)
  MoveL 3612 to (496.46, 561.58, 64) mm, rotated rx -180 ry 0 rz 160 deg; joints [13.928, 69.522, -8.192, -142.524, 66.542, 163.028]
  Set speed (17.7 mm/s)
  Call Extruder(1342.33653)
  MoveL 3613 to (493.94, 561.39, 64) mm, rotated rx -180 ry 0 rz 160 deg; joints [13.98, 69.147, -7.354, -142.59, 66.924, 163.312]
  Set speed (17.7 mm/s)
  Call Extruder(1350.31998)
  MoveL 3614 to (491.45, 561.09, 64) mm, rotated rx 180 ry 0 rz 160 deg; joints [14.02, 68.779, -6.531, -142.665, 67.297, 163.596]
  Set speed (17.7 mm/s)
  Call Extruder(1358.26434)
  MoveL 3615 to (488.99, 560.7, 64) mm, rotated rx 180 ry 0 rz 160 deg; joints [14.047, 68.416, -5.717, -142.751, 67.664, 163.882]
  Call Extruder(1366.51474)
  MoveL 3616 to (486.46, 560.18, 64) mm, rotated rx 180 ry 0 rz 160 deg; joints [14.061, 68.044, -4.877, -142.851, 68.04, 164.181]
  Set speed (17.7 mm/s)
  Call Extruder(1370.49125)
  MoveL 3617 to (485.25, 559.89, 64) mm, rotated rx -180 ry 0 rz 160 deg; joints [14.063, 67.867, -4.476, -142.903, 68.219, 164.326]
  Call Extruder(1374.51721)
  MoveL 3618 to (484.03, 559.58, 64) mm, rotated rx -180 ry 0 rz 160 deg; joints [14.063, 67.688, -4.072, -142.958, 68.399, 164.473]
  Call Extruder(1378.52277)
  MoveL 3619 to (482.82, 559.24, 64) mm, rotated rx -180 ry 0 rz 160 deg; joints [14.057, 67.512, -3.672, -143.016, 68.577, 164.62]
  Set speed (17.7 mm/s)
  Call Extruder(1382.46385)
  MoveL 3620 to (481.64, 558.89, 64) mm, rotated rx 180 ry 0 rz 160 deg; joints [14.051, 67.34, -3.281, -143.075, 68.75, 164.764]
  Set speed (17.7 mm/s)
  Call Extruder(1386.57112)
  MoveL 3621 to (480.42, 558.49, 64) mm, rotated rx 180 ry 0 rz 160 deg; joints [14.039, 67.162, -2.875, -143.14, 68.929, 164.915]
  Set speed (17.7 mm/s)
  Call Extruder(1390.55055)
  MoveL 3622 to (479.24, 558.09, 64) mm, rotated rx 180 ry 0 rz 160 deg; joints [14.025, 66.992, -2.485, -143.204, 69.101, 165.061]
  Set speed (17.7 mm/s)
  Call Extruder(1394.67318)
  MoveL 3623 to (478.03, 557.63, 64) mm, rotated rx -180 ry 0 rz 160 deg; joints [14.006, 66.816, -2.083, -143.275, 69.278, 165.212]
  Set speed (17.7 mm/s)
  Call Extruder(1398.86426)
  MoveL 3624 to (476.81, 557.16, 64) mm, rotated rx -180 ry 0 rz 160 deg; joints [13.985, 66.639, -1.678, -143.349, 69.455, 165.366]
  Call Extruder(1402.73183)
  MoveL 3625 to (475.69, 556.69, 64) mm, rotated rx 180 ry 0 rz 160 deg; joints [13.961, 66.478, -1.307, -143.421, 69.617, 165.508]
  Set speed (17.7 mm/s)
  Call Extruder(1406.68057)
  MoveL 3626 to (474.56, 556.2, 64) mm, rotated rx 180 ry 0 rz 160 deg; joints [13.934, 66.315, -0.931, -143.495, 69.782, 165.653]
  Set speed (17.7 mm/s)
  Call Extruder(1410.73544)
  MoveL 3627 to (473.41, 555.66, 64) mm, rotated rx -180 ry 0 rz 160 deg; joints [13.902, 66.148, -0.547, -143.576, 69.949, 165.802]
  Set speed (17.7 mm/s)
  Call Extruder(1414.70483)
  MoveL 3628 to (472.29, 555.11, 64) mm, rotated rx -180 ry 0 rz 160 deg; joints [13.867, 65.988, -0.176, -143.657, 70.11, 165.947]
  Call Extruder(1418.75289)
  MoveL 3629 to (471.16, 554.53, 64) mm, rotated rx -180 ry 0 rz 160 deg; joints [13.828, 65.825, 0.2, -143.743, 70.273, 166.095]
  Set speed (17.7 mm/s)
  Call Extruder(1423.51412)
  MoveL 3630 to (469.85, 553.82, 64) mm, rotated rx -180 ry 0 rz 160 deg; joints [13.777, 65.637, 0.638, -143.848, 70.462, 166.269]
  Set speed (17.7 mm/s)
  Call Extruder(1426.78002)
  MoveL 3631 to (468.96, 553.31, 64) mm, rotated rx 180 ry 0 rz 160 deg; joints [13.74, 65.509, 0.935, -143.922, 70.59, 166.388]
  Set speed (17.7 mm/s)
  Call Extruder(1430.83262)
  MoveL 3632 to (467.87, 552.66, 64) mm, rotated rx 180 ry 0 rz 160 deg; joints [13.69, 65.353, 1.301, -144.016, 70.747, 166.535]
  Set speed (17.7 mm/s)
  Call Extruder(1434.86482)
  MoveL 3633 to (466.8, 551.99, 64) mm, rotated rx 180 ry 0 rz 160 deg; joints [13.637, 65.199, 1.66, -144.112, 70.901, 166.681]
  Set speed (17.7 mm/s)
  Call Extruder(1438.82835)
  MoveL 3634 to (465.76, 551.31, 64) mm, rotated rx 180 ry 0 rz 160 deg; joints [13.582, 65.049, 2.01, -144.21, 71.051, 166.824]
  Set speed (17.7 mm/s)
  Call Extruder(1442.91652)
  MoveL 3635 to (464.7, 550.59, 64) mm, rotated rx -180 ry 0 rz 160 deg; joints [13.521, 64.898, 2.366, -144.314, 71.203, 166.97]
  Set speed (17.7 mm/s)
  Call Extruder(1446.91650)
  MoveL 3636 to (463.68, 549.86, 64) mm, rotated rx -180 ry 0 rz 160 deg; joints [13.457, 64.751, 2.71, -144.418, 71.35, 167.113]
  Set speed (17.7 mm/s)
  Call Extruder(1450.96243)
  MoveL 3637 to (462.66, 549.1, 64) mm, rotated rx 180 ry 0 rz 160 deg; joints [13.389, 64.605, 3.054, -144.526, 71.496, 167.256]
  Set speed (17.7 mm/s)
  Call Extruder(1454.91285)
  MoveL 3638 to (461.68, 548.34, 64) mm, rotated rx -180 ry 0 rz 160 deg; joints [13.32, 64.465, 3.385, -144.635, 71.636, 167.395]
  Set speed (17.7 mm/s)
  Call Extruder(1458.99965)
  MoveL 3639 to (460.69, 547.54, 64) mm, rotated rx 180 ry 0 rz 160 deg; joints [13.245, 64.322, 3.723, -144.749, 71.779, 167.539]
  Set speed (17.7 mm/s)
  Call Extruder(1463.04809)
  MoveL 3640 to (459.72, 546.72, 64) mm, rotated rx 180 ry 0 rz 160 deg; joints [13.166, 64.183, 4.053, -144.866, 71.918, 167.679]
  Set speed (17.7 mm/s)
  Call Extruder(1467.00098)
  MoveL 3641 to (458.79, 545.9, 64) mm, rotated rx -180 ry 0 rz 160 deg; joints [13.086, 64.049, 4.37, -144.983, 72.051, 167.816]
  Set speed (17.7 mm/s)
  Call Extruder(1471.01655)
  MoveL 3642 to (457.86, 545.05, 64) mm, rotated rx -180 ry 0 rz 160 deg; joints [13.001, 63.916, 4.687, -145.104, 72.184, 167.953]
  Set speed (17.7 mm/s)
  Call Extruder(1474.23497)
  MoveL 3643 to (457.13, 544.36, 64) mm, rotated rx -180 ry 0 rz 160 deg; joints [12.931, 63.811, 4.939, -145.202, 72.289, 168.063]
  Set speed (17.7 mm/s)
  Call Extruder(1479.31345)
  MoveL 3644 to (456, 543.23, 64) mm, rotated rx 180 ry 0 rz 160 deg; joints [12.815, 63.648, 5.328, -145.363, 72.451, 168.234]
  Set speed (17.7 mm/s)
  Call Extruder(1483.16580)
  MoveL 3645 to (455.16, 542.36, 64) mm, rotated rx -180 ry 0 rz 160 deg; joints [12.723, 63.527, 5.617, -145.487, 72.571, 168.362]
  Call Extruder(1487.11031)
  MoveL 3646 to (454.32, 541.45, 64) mm, rotated rx 180 ry 0 rz 160 deg; joints [12.626, 63.406, 5.908, -145.617, 72.692, 168.493]
  Set speed (17.7 mm/s)
  Call Extruder(1491.19591)
  MoveL 3647 to (453.47, 540.5, 64) mm, rotated rx 180 ry 0 rz 160 deg; joints [12.522, 63.283, 6.204, -145.753, 72.814, 168.627]
  Set speed (17.7 mm/s)
  Call Extruder(1495.18276)
  MoveL 3648 to (452.66, 539.54, 64) mm, rotated rx -180 ry 0 rz 160 deg; joints [12.418, 63.166, 6.487, -145.89, 72.931, 168.756]
  Call Extruder(1499.24676)
  MoveL 3649 to (451.85, 538.56, 64) mm, rotated rx -180 ry 0 rz 160 deg; joints [12.308, 63.048, 6.77, -146.031, 73.047, 168.886]
  Call Extruder(1503.28876)
  MoveL 3650 to (451.07, 537.56, 64) mm, rotated rx 180 ry 0 rz 160 deg; joints [12.195, 62.935, 7.045, -146.174, 73.159, 169.013]
  Set speed (17.7 mm/s)
  Call Extruder(1507.27611)
  MoveL 3651 to (450.32, 536.57, 64) mm, rotated rx -180 ry 0 rz 160 deg; joints [12.08, 62.825, 7.311, -146.318, 73.267, 169.138]
  Set speed (17.7 mm/s)
  Call Extruder(1511.33033)
  MoveL 3652 to (449.58, 535.53, 64) mm, rotated rx -180 ry 0 rz 160 deg; joints [11.96, 62.716, 7.575, -146.466, 73.374, 169.263]
  Set speed (17.7 mm/s)
  Call Extruder(1515.31430)
  MoveL 3653 to (448.87, 534.5, 64) mm, rotated rx 180 ry 0 rz 160 deg; joints [11.839, 62.612, 7.829, -146.615, 73.476, 169.384]
  Call Extruder(1519.45266)
  MoveL 3654 to (448.15, 533.42, 64) mm, rotated rx -180 ry 0 rz 160 deg; joints [11.71, 62.506, 8.086, -146.772, 73.579, 169.509]
  Set speed (17.7 mm/s)
  Call Extruder(1523.35069)
  MoveL 3655 to (447.5, 532.39, 64) mm, rotated rx -180 ry 0 rz 160 deg; joints [11.586, 62.41, 8.322, -146.922, 73.674, 169.624]
  Call Extruder(1527.37566)
  MoveL 3656 to (446.85, 531.31, 64) mm, rotated rx -180 ry 0 rz 160 deg; joints [11.454, 62.313, 8.559, -147.079, 73.768, 169.741]
  Set speed (17.7 mm/s)
  Call Extruder(1531.52863)
  MoveL 3657 to (446.2, 530.18, 64) mm, rotated rx -180 ry 0 rz 160 deg; joints [11.315, 62.216, 8.797, -147.243, 73.861, 169.86]
  Set speed (17.7 mm/s)
  Call Extruder(1535.43515)
  MoveL 3658 to (445.61, 529.11, 64) mm, rotated rx 180 ry 0 rz 160 deg; joints [11.182, 62.127, 9.014, -147.4, 73.946, 169.971]
  Set speed (17.7 mm/s)
  Call Extruder(1539.49791)
  MoveL 3659 to (445.02, 527.98, 64) mm, rotated rx 180 ry 0 rz 160 deg; joints [11.041, 62.038, 9.234, -147.565, 74.032, 170.084]
  Call Extruder(1543.47866)
  MoveL 3660 to (444.47, 526.86, 64) mm, rotated rx -180 ry 0 rz 160 deg; joints [10.899, 61.953, 9.442, -147.729, 74.112, 170.192]
  Set speed (17.7 mm/s)
  Call Extruder(1547.64280)
  MoveL 3661 to (443.92, 525.68, 64) mm, rotated rx 180 ry 0 rz 160 deg; joints [10.748, 61.868, 9.651, -147.903, 74.192, 170.304]
  Set speed (17.7 mm/s)
  Call Extruder(1551.59336)
  MoveL 3662 to (443.41, 524.55, 64) mm, rotated rx -180 ry 0 rz 160 deg; joints [10.603, 61.79, 9.846, -148.069, 74.265, 170.408]
  Set speed (17.7 mm/s)
  Call Extruder(1558.93923)
  MoveL 3663 to (442.53, 522.43, 64) mm, rotated rx 180 ry 0 rz 160 deg; joints [10.325, 61.652, 10.187, -148.383, 74.393, 170.596]
  Set speed (17.6 mm/s)
  Call Extruder(1563.76664)
  MoveL 3664 to (442.01, 521.01, 64) mm, rotated rx -180 ry 0 rz 160 deg; joints [10.138, 61.567, 10.397, -148.593, 74.469, 170.715]
  Set speed (17.7 mm/s)
  Call Extruder(1567.73704)
  MoveL 3665 to (441.59, 519.84, 64) mm, rotated rx 180 ry 0 rz 160 deg; joints [9.982, 61.5, 10.564, -148.767, 74.53, 170.812]
  Call Extruder(0.00000)
  Set speed (17.7 mm/s)
  Call Extruder(8.11575)
  MoveL 3666 to (440.82, 517.42, 64) mm, rotated rx -180 ry 0 rz 160 deg; joints [9.656, 61.372, 10.882, -149.128, 74.641, 171.002]
  Set speed (17.7 mm/s)
  Call Extruder(12.14859)
  MoveL 3667 to (440.48, 516.2, 64) mm, rotated rx -180 ry 0 rz 160 deg; joints [9.49, 61.314, 11.027, -149.31, 74.69, 171.093]
  Set speed (17.7 mm/s)
  Call Extruder(16.10375)
  MoveL 3668 to (440.17, 515, 64) mm, rotated rx 180 ry 0 rz 160 deg; joints [9.327, 61.259, 11.165, -149.489, 74.736, 171.181]
  Call Extruder(20.19222)
  MoveL 3669 to (439.88, 513.76, 64) mm, rotated rx -180 ry 0 rz 160 deg; joints [9.155, 61.206, 11.297, -149.676, 74.778, 171.269]
  Set speed (17.7 mm/s)
  Call Extruder(24.13653)
  MoveL 3670 to (439.61, 512.55, 64) mm, rotated rx 180 ry 0 rz 160 deg; joints [8.988, 61.157, 11.42, -149.857, 74.816, 171.352]
  Set speed (17.7 mm/s)
  Call Extruder(32.30771)
  MoveL 3671 to (439.14, 510.03, 64) mm, rotated rx -180 ry 0 rz 160 deg; joints [8.636, 61.066, 11.648, -150.237, 74.883, 171.518]
  Set speed (17.7 mm/s)
  Call Extruder(40.35460)
  MoveL 3672 to (438.78, 507.54, 64) mm, rotated rx -180 ry 0 rz 160 deg; joints [8.283, 60.988, 11.843, -150.614, 74.933, 171.672]
  Set speed (17.7 mm/s)
  Call Extruder(48.39644)
  MoveL 3673 to (438.52, 505.03, 64) mm, rotated rx -180 ry 0 rz 160 deg; joints [7.925, 60.923, 12.006, -150.993, 74.968, 171.817]
  Set speed (17.7 mm/s)
  Call Extruder(56.29267)
  MoveL 3674 to (438.37, 502.56, 64) mm, rotated rx 180 ry 0 rz 160 deg; joints [7.57, 60.872, 12.135, -151.368, 74.986, 171.95]
  Call Extruder(64.41839)
  MoveL 3675 to (438.32, 500.01, 64) mm, rotated rx 180 ry 0 rz 160 deg; joints [7.201, 60.832, 12.237, -151.754, 74.988, 172.078]
  Set speed (17.7 mm/s)
  Call Extruder(71.74111)
  MoveL 3676 to (438.35, 497.72, 64) mm, rotated rx -180 ry 0 rz 160 deg; joints [6.866, 60.806, 12.302, -152.102, 74.977, 172.186]
  Set speed (17.7 mm/s)
  Call Extruder(78.90339)
  MoveL 3677 to (438.48, 495.48, 64) mm, rotated rx 180 ry 0 rz 160 deg; joints [6.537, 60.792, 12.338, -152.442, 74.952, 172.284]
  Set speed (17.7 mm/s)
  Call Extruder(86.16086)
  MoveL 3678 to (438.69, 493.21, 64) mm, rotated rx -180 ry 0 rz 160 deg; joints [6.203, 60.787, 12.35, -152.786, 74.914, 172.377]
  Call Extruder(93.40935)
  MoveL 3679 to (438.98, 490.96, 64) mm, rotated rx 180 ry 0 rz 160 deg; joints [5.87, 60.793, 12.336, -153.127, 74.862, 172.462]
  Set speed (17.7 mm/s)
  Call Extruder(100.74127)
  MoveL 3680 to (439.36, 488.69, 64) mm, rotated rx 180 ry 0 rz 160 deg; joints [5.533, 60.809, 12.295, -153.47, 74.796, 172.541]
  Call Extruder(107.83794)
  MoveL 3681 to (439.81, 486.52, 64) mm, rotated rx -180 ry 0 rz 160 deg; joints [5.209, 60.834, 12.231, -153.798, 74.719, 172.611]
  Set speed (17.7 mm/s)
  Call Extruder(115.14144)
  MoveL 3682 to (440.35, 484.29, 64) mm, rotated rx 180 ry 0 rz 160 deg; joints [4.878, 60.871, 12.139, -154.133, 74.627, 172.675]
  Set speed (17.7 mm/s)
  Call Extruder(122.38871)
  MoveL 3683 to (440.97, 482.11, 64) mm, rotated rx -180 ry 0 rz 160 deg; joints [4.551, 60.917, 12.022, -154.46, 74.522, 172.733]
  Set speed (17.7 mm/s)
  Call Extruder(129.57460)
  MoveL 3684 to (441.66, 479.96, 64) mm, rotated rx -180 ry 0 rz 160 deg; joints [4.231, 60.974, 11.88, -154.78, 74.405, 172.783]
  Call Extruder(136.95879)
  MoveL 3685 to (442.45, 477.79, 64) mm, rotated rx 180 ry 0 rz 160 deg; joints [3.906, 61.042, 11.709, -155.102, 74.271, 172.829]
  Call Extruder(144.20691)
  MoveL 3686 to (443.31, 475.68, 64) mm, rotated rx -180 ry 0 rz 160 deg; joints [3.591, 61.119, 11.516, -155.413, 74.126, 172.866]
  Set speed (17.7 mm/s)
  Call Extruder(151.35641)
  MoveL 3687 to (444.23, 473.64, 64) mm, rotated rx -180 ry 0 rz 160 deg; joints [3.286, 61.204, 11.301, -155.712, 73.971, 172.897]
  Set speed (17.7 mm/s)
  Call Extruder(158.68987)
  MoveL 3688 to (445.25, 471.58, 64) mm, rotated rx 180 ry 0 rz 160 deg; joints [2.98, 61.302, 11.056, -156.012, 73.799, 172.923]
  Set speed (17.7 mm/s)
  Call Extruder(165.77468)
  MoveL 3689 to (446.31, 469.63, 64) mm, rotated rx -180 ry 0 rz 160 deg; joints [2.69, 61.407, 10.796, -156.293, 73.621, 172.941]
  Set speed (17.7 mm/s)
  Call Extruder(173.13299)
  MoveL 3690 to (447.48, 467.64, 64) mm, rotated rx 180 ry 0 rz 160 deg; joints [2.396, 61.525, 10.501, -156.576, 73.423, 172.954]
  Call Extruder(180.34598)
  MoveL 3691 to (448.7, 465.74, 64) mm, rotated rx 180 ry 0 rz 160 deg; joints [2.115, 61.651, 10.19, -156.845, 73.218, 172.961]
  Call Extruder(187.43961)
  MoveL 3692 to (449.97, 463.91, 64) mm, rotated rx -180 ry 0 rz 160 deg; joints [1.846, 61.784, 9.86, -157.101, 73.004, 172.961]
  Set speed (17.7 mm/s)
  Call Extruder(194.92373)
  MoveL 3693 to (451.38, 462.04, 64) mm, rotated rx -180 ry 0 rz 160 deg; joints [1.572, 61.934, 9.49, -157.359, 72.767, 172.956]
  Call Extruder(202.02603)
  MoveL 3694 to (452.78, 460.31, 64) mm, rotated rx 180 ry 0 rz 160 deg; joints [1.32, 62.086, 9.116, -157.595, 72.531, 172.945]
  Set speed (17.7 mm/s)
  Call Extruder(209.33385)
  MoveL 3695 to (454.29, 458.58, 64) mm, rotated rx 180 ry 0 rz 160 deg; joints [1.07, 62.251, 8.71, -157.826, 72.278, 172.928]
  Set speed (17.7 mm/s)
  Call Extruder(216.66129)
  MoveL 3696 to (455.86, 456.91, 64) mm, rotated rx -180 ry 0 rz 160 deg; joints [0.83, 62.426, 8.281, -158.046, 72.013, 172.905]
  Call Extruder(223.71689)
  MoveL 3697 to (457.43, 455.36, 64) mm, rotated rx 180 ry 0 rz 160 deg; joints [0.608, 62.604, 7.847, -158.247, 71.748, 172.877]
  Set speed (17.7 mm/s)
  Call Extruder(231.06352)
  MoveL 3698 to (459.13, 453.8, 64) mm, rotated rx 180 ry 0 rz 160 deg; joints [0.387, 62.798, 7.376, -158.444, 71.463, 172.841]
  Set speed (17.7 mm/s)
  Call Extruder(238.12920)
  MoveL 3699 to (460.82, 452.36, 64) mm, rotated rx -180 ry 0 rz 160 deg; joints [0.184, 62.993, 6.903, -158.621, 71.179, 172.802]
  Set speed (17.7 mm/s)
  Call Extruder(245.99854)
  MoveL 3700 to (462.75, 450.83, 64) mm, rotated rx -180 ry 0 rz 160 deg; joints [-0.029, 63.22, 6.355, -158.805, 70.853, 172.752]
  Set speed (17.7 mm/s)
  Call Extruder(252.33579)
  MoveL 3701 to (464.35, 449.66, 64) mm, rotated rx 180 ry 0 rz 160 deg; joints [-0.192, 63.41, 5.899, -158.942, 70.584, 172.706]
  Set speed (17.7 mm/s)
  Call Extruder(259.95298)
  MoveL 3702 to (466.32, 448.32, 64) mm, rotated rx -180 ry 0 rz 160 deg; joints [-0.376, 63.646, 5.332, -159.094, 70.252, 172.646]
  Set speed (17.7 mm/s)
  Call Extruder(267.38150)
  MoveL 3703 to (468.3, 447.08, 64) mm, rotated rx -180 ry 0 rz 160 deg; joints [-0.543, 63.885, 4.761, -159.228, 69.92, 172.58]
  Set speed (17.7 mm/s)
  Call Extruder(274.63255)
  MoveL 3704 to (470.27, 445.95, 64) mm, rotated rx 180 ry 0 rz 160 deg; joints [-0.695, 64.126, 4.187, -159.345, 69.589, 172.51]
  Set speed (17.7 mm/s)
  Call Extruder(282.74772)
  MoveL 3705 to (472.51, 444.77, 64) mm, rotated rx 180 ry 0 rz 160 deg; joints [-0.851, 64.405, 3.526, -159.46, 69.211, 172.425]
  Set speed (17.7 mm/s)
  Call Extruder(289.14680)
  MoveL 3706 to (474.32, 443.91, 64) mm, rotated rx 180 ry 0 rz 160 deg; joints [-0.964, 64.632, 2.991, -159.538, 68.907, 172.352]
  Set speed (17.7 mm/s)
  Call Extruder(296.12587)
  MoveL 3707 to (476.33, 443.04, 64) mm, rotated rx 180 ry 0 rz 160 deg; joints [-1.077, 64.886, 2.394, -159.612, 68.57, 172.267]
  Call Extruder(303.49803)
  MoveL 3708 to (478.48, 442.19, 64) mm, rotated rx 180 ry 0 rz 160 deg; joints [-1.185, 65.16, 1.75, -159.676, 68.209, 172.171]
  Call Extruder(310.64970)
  MoveL 3709 to (480.59, 441.45, 64) mm, rotated rx -180 ry 0 rz 160 deg; joints [-1.279, 65.434, 1.111, -159.725, 67.854, 172.072]
  Set speed (17.7 mm/s)
  Call Extruder(317.97503)
  MoveL 3710 to (482.79, 440.77, 64) mm, rotated rx 180 ry 0 rz 160 deg; joints [-1.363, 65.72, 0.444, -159.76, 67.485, 171.964]
  Set speed (17.7 mm/s)
  Call Extruder(325.13582)
  MoveL 3711 to (484.95, 440.18, 64) mm, rotated rx -180 ry 0 rz 160 deg; joints [-1.433, 66.007, -0.219, -159.782, 67.121, 171.852]
  Set speed (17.7 mm/s)
  Call Extruder(332.53379)
  MoveL 3712 to (487.21, 439.66, 64) mm, rotated rx -180 ry 0 rz 160 deg; joints [-1.494, 66.308, -0.916, -159.79, 66.742, 171.729]
  Set speed (17.7 mm/s)
  Call Extruder(339.72115)
  MoveL 3713 to (489.42, 439.23, 64) mm, rotated rx 180 ry 0 rz 160 deg; joints [-1.542, 66.607, -1.603, -159.783, 66.37, 171.603]
  Set speed (17.7 mm/s)
  Call Extruder(346.69068)
  MoveL 3714 to (491.58, 438.89, 64) mm, rotated rx 180 ry 0 rz 160 deg; joints [-1.579, 66.901, -2.278, -159.764, 66.008, 171.475]
  Set speed (17.7 mm/s)
  Call Extruder(354.26599)
  MoveL 3715 to (493.94, 438.61, 64) mm, rotated rx 180 ry 0 rz 160 deg; joints [-1.606, 67.227, -3.022, -159.729, 65.611, 171.329]
  Set speed (17.7 mm/s)
  Call Extruder(361.51893)
  MoveL 3716 to (496.2, 438.43, 64) mm, rotated rx 180 ry 0 rz 160 deg; joints [-1.621, 67.543, -3.741, -159.681, 65.231, 171.182]
  Set speed (17.7 mm/s)
  Call Extruder(368.85059)
  MoveL 3717 to (498.5, 438.33, 64) mm, rotated rx 180 ry 0 rz 160 deg; joints [-1.626, 67.867, -4.477, -159.62, 64.845, 171.026]
  Set speed (17.7 mm/s)
  Call Extruder(376.03099)
  MoveL 3718 to (500.75, 438.32, 64) mm, rotated rx 180 ry 0 rz 160 deg; joints [-1.619, 68.189, -5.204, -159.546, 64.465, 170.867]
  Set speed (17.7 mm/s)
  Call Extruder(383.13923)
  MoveL 3719 to (502.98, 438.39, 64) mm, rotated rx 180 ry 0 rz 160 deg; joints [-1.603, 68.511, -5.93, -159.46, 64.09, 170.702]
  Call Extruder(390.51309)
  MoveL 3720 to (505.28, 438.54, 64) mm, rotated rx 180 ry 0 rz 160 deg; joints [-1.575, 68.848, -6.687, -159.357, 63.702, 170.524]
  Set speed (17.7 mm/s)
  Call Extruder(397.84152)
  MoveL 3721 to (507.57, 438.78, 64) mm, rotated rx 180 ry 0 rz 160 deg; joints [-1.537, 69.187, -7.444, -159.241, 63.316, 170.34]
  Set speed (17.7 mm/s)
  Call Extruder(404.91505)
  MoveL 3722 to (509.76, 439.09, 64) mm, rotated rx 180 ry 0 rz 160 deg; joints [-1.491, 69.516, -8.178, -159.118, 62.946, 170.156]
  Set speed (17.7 mm/s)
  Call Extruder(412.30867)
  MoveL 3723 to (512.05, 439.5, 64) mm, rotated rx -180 ry 0 rz 160 deg; joints [-1.433, 69.862, -8.947, -158.975, 62.561, 169.956]
  Set speed (17.7 mm/s)
  Call Extruder(419.49856)
  MoveL 3724 to (514.25, 439.98, 64) mm, rotated rx -180 ry 0 rz 160 deg; joints [-1.367, 70.2, -9.697, -158.824, 62.189, 169.755]
  Call Extruder(426.64755)
  MoveL 3725 to (516.42, 440.54, 64) mm, rotated rx -180 ry 0 rz 160 deg; joints [-1.292, 70.538, -10.443, -158.662, 61.822, 169.548]
  Set speed (17.7 mm/s)
  Call Extruder(433.98030)
  MoveL 3726 to (518.62, 441.19, 64) mm, rotated rx -180 ry 0 rz 160 deg; joints [-1.206, 70.886, -11.209, -158.483, 61.448, 169.329]
  Set speed (17.7 mm/s)
  Call Extruder(441.28921)
  MoveL 3727 to (520.8, 441.93, 64) mm, rotated rx 180 ry 0 rz 160 deg; joints [-1.111, 71.233, -11.97, -158.293, 61.081, 169.104]
  Set speed (17.7 mm/s)
  Call Extruder(448.43280)
  MoveL 3728 to (522.89, 442.72, 64) mm, rotated rx 180 ry 0 rz 160 deg; joints [-1.01, 71.572, -12.713, -158.096, 60.725, 168.877]
  Set speed (17.7 mm/s)
  Call Extruder(455.76980)
  MoveL 3729 to (525.01, 443.61, 64) mm, rotated rx -180 ry 0 rz 160 deg; joints [-0.897, 71.92, -13.472, -157.882, 60.366, 168.637]
  Call Extruder(462.96365)
  MoveL 3730 to (527.06, 444.56, 64) mm, rotated rx 180 ry 0 rz 160 deg; joints [-0.779, 72.261, -14.214, -157.662, 60.019, 168.397]
  Set speed (17.7 mm/s)
  Call Extruder(470.10483)
  MoveL 3731 to (529.05, 445.58, 64) mm, rotated rx 180 ry 0 rz 160 deg; joints [-0.654, 72.598, -14.944, -157.433, 59.68, 168.151]
  Call Extruder(477.50712)
  MoveL 3732 to (531.08, 446.71, 64) mm, rotated rx -180 ry 0 rz 160 deg; joints [-0.516, 72.945, -15.696, -157.185, 59.336, 167.891]
  Set speed (17.7 mm/s)
  Call Extruder(484.65795)
  MoveL 3733 to (532.99, 447.88, 64) mm, rotated rx -180 ry 0 rz 160 deg; joints [-0.376, 73.278, -16.414, -156.935, 59.01, 167.634]
  Set speed (17.7 mm/s)
  Call Extruder(491.98460)
  MoveL 3734 to (534.91, 449.14, 64) mm, rotated rx 180 ry 0 rz 160 deg; joints [-0.225, 73.616, -17.143, -156.67, 58.684, 167.365]
  Set speed (17.7 mm/s)
  Call Extruder(499.14816)
  MoveL 3735 to (536.74, 450.45, 64) mm, rotated rx 180 ry 0 rz 160 deg; joints [-0.07, 73.944, -17.846, -156.402, 58.374, 167.098]
  Set speed (17.7 mm/s)
  Call Extruder(506.39876)
  MoveL 3736 to (538.54, 451.83, 64) mm, rotated rx -180 ry 0 rz 160 deg; joints [0.093, 74.271, -18.548, -156.121, 58.068, 166.822]
  Set speed (17.7 mm/s)
  Call Extruder(513.63589)
  MoveL 3737 to (540.28, 453.28, 64) mm, rotated rx 180 ry 0 rz 160 deg; joints [0.262, 74.594, -19.238, -155.833, 57.771, 166.542]
  Call Extruder(520.95921)
  MoveL 3738 to (541.99, 454.82, 64) mm, rotated rx 180 ry 0 rz 160 deg; joints [0.44, 74.915, -19.924, -155.534, 57.481, 166.255]
  Call Extruder(528.16880)
  MoveL 3739 to (543.62, 456.38, 64) mm, rotated rx -180 ry 0 rz 160 deg; joints [0.621, 75.226, -20.586, -155.231, 57.205, 165.969]
  Set speed (17.7 mm/s)
  Call Extruder(532.14467)
  MoveL 3740 to (544.49, 457.27, 64) mm, rotated rx -180 ry 0 rz 160 deg; joints [0.723, 75.395, -20.944, -155.062, 57.058, 165.81]
  Set speed (17.7 mm/s)
  Call Extruder(536.10256)
  MoveL 3741 to (545.34, 458.18, 64) mm, rotated rx 180 ry 0 rz 160 deg; joints [0.826, 75.561, -21.297, -154.891, 56.915, 165.651]
  Call Extruder(540.19728)
  MoveL 3742 to (546.2, 459.13, 64) mm, rotated rx 180 ry 0 rz 160 deg; joints [0.935, 75.731, -21.656, -154.713, 56.77, 165.485]
  Set speed (17.7 mm/s)
  Call Extruder(544.13499)
  MoveL 3743 to (547.01, 460.06, 64) mm, rotated rx -180 ry 0 rz 160 deg; joints [1.041, 75.892, -21.998, -154.539, 56.634, 165.325]
  Set speed (17.7 mm/s)
  Call Extruder(548.16663)
  MoveL 3744 to (547.82, 461.03, 64) mm, rotated rx -180 ry 0 rz 160 deg; joints [1.151, 76.055, -22.342, -154.36, 56.498, 165.161]
  Call Extruder(552.25885)
  MoveL 3745 to (548.62, 462.04, 64) mm, rotated rx 180 ry 0 rz 160 deg; joints [1.265, 76.217, -22.686, -154.176, 56.364, 164.994]
  Call Extruder(556.22308)
  MoveL 3746 to (549.37, 463.02, 64) mm, rotated rx -180 ry 0 rz 160 deg; joints [1.376, 76.372, -23.013, -153.996, 56.239, 164.832]
  Set speed (17.7 mm/s)
  Call Extruder(560.34596)
  MoveL 3747 to (550.14, 464.07, 64) mm, rotated rx 180 ry 0 rz 160 deg; joints [1.494, 76.531, -23.347, -153.808, 56.111, 164.663]
  Set speed (17.7 mm/s)
  Call Extruder(564.25349)
  MoveL 3748 to (550.84, 465.07, 64) mm, rotated rx 180 ry 0 rz 160 deg; joints [1.606, 76.679, -23.659, -153.629, 55.994, 164.502]
  Set speed (17.7 mm/s)
  Call Extruder(568.31395)
  MoveL 3749 to (551.55, 466.12, 64) mm, rotated rx 180 ry 0 rz 160 deg; joints [1.725, 76.829, -23.976, -153.441, 55.877, 164.336]
  Call Extruder(571.70237)
  MoveL 3750 to (552.13, 467.02, 64) mm, rotated rx -180 ry 0 rz 160 deg; joints [1.825, 76.953, -24.235, -153.283, 55.783, 164.197]
  Set speed (17.7 mm/s)
  Call Extruder(576.43739)
  MoveL 3751 to (552.91, 468.28, 64) mm, rotated rx -180 ry 0 rz 160 deg; joints [1.966, 77.122, -24.591, -153.061, 55.656, 164.003]
  Set speed (17.7 mm/s)
  Call Extruder(580.44693)
  MoveL 3752 to (553.54, 469.36, 64) mm, rotated rx 180 ry 0 rz 160 deg; joints [2.087, 77.262, -24.884, -152.873, 55.552, 163.838]
  Set speed (17.7 mm/s)
  Call Extruder(584.42205)
  MoveL 3753 to (554.15, 470.45, 64) mm, rotated rx 180 ry 0 rz 160 deg; joints [2.208, 77.397, -25.167, -152.685, 55.454, 163.676]
  Set speed (17.7 mm/s)
  Call Extruder(588.48894)
  MoveL 3754 to (554.75, 471.58, 64) mm, rotated rx -180 ry 0 rz 160 deg; joints [2.333, 77.532, -25.45, -152.492, 55.358, 163.511]
  Call Extruder(592.48613)
  MoveL 3755 to (555.32, 472.69, 64) mm, rotated rx -180 ry 0 rz 160 deg; joints [2.457, 77.662, -25.722, -152.302, 55.268, 163.348]
  Set speed (17.7 mm/s)
  Call Extruder(596.48575)
  MoveL 3756 to (555.86, 473.82, 64) mm, rotated rx 180 ry 0 rz 160 deg; joints [2.582, 77.787, -25.985, -152.112, 55.182, 163.187]
  Set speed (17.7 mm/s)
  Call Extruder(600.57557)
  MoveL 3757 to (556.39, 474.99, 64) mm, rotated rx 180 ry 0 rz 160 deg; joints [2.711, 77.912, -26.246, -151.917, 55.1, 163.023]
  Set speed (17.7 mm/s)
  Call Extruder(604.62401)
  MoveL 3758 to (556.88, 476.16, 64) mm, rotated rx -180 ry 0 rz 160 deg; joints [2.84, 78.031, -26.494, -151.723, 55.024, 162.863]
  Set speed (17.7 mm/s)
  Call Extruder(608.74837)
  MoveL 3759 to (557.38, 477.35, 64) mm, rotated rx -180 ry 0 rz 160 deg; joints [2.972, 78.15, -26.743, -151.526, 54.948, 162.699]
  Set speed (17.7 mm/s)
  Call Extruder(612.68746)
  MoveL 3760 to (557.81, 478.51, 64) mm, rotated rx 180 ry 0 rz 160 deg; joints [3.1, 78.258, -26.968, -151.338, 54.884, 162.545]
  Set speed (17.7 mm/s)
  Call Extruder(616.65325)
  MoveL 3761 to (558.24, 479.67, 64) mm, rotated rx -180 ry 0 rz 160 deg; joints [3.229, 78.365, -27.191, -151.149, 54.821, 162.391]
  Set speed (17.7 mm/s)
  Call Extruder(620.76877)
  MoveL 3762 to (558.65, 480.89, 64) mm, rotated rx 180 ry 0 rz 160 deg; joints [3.363, 78.469, -27.408, -150.953, 54.763, 162.233]
  Set speed (17.7 mm/s)
  Call Extruder(624.93290)
  MoveL 3763 to (559.04, 482.13, 64) mm, rotated rx -180 ry 0 rz 160 deg; joints [3.5, 78.573, -27.624, -150.755, 54.707, 162.074]
  Call Extruder(628.79515)
  MoveL 3764 to (559.38, 483.3, 64) mm, rotated rx 180 ry 0 rz 160 deg; joints [3.628, 78.662, -27.81, -150.572, 54.662, 161.93]
  Call Extruder(632.64312)
  MoveL 3765 to (559.69, 484.46, 64) mm, rotated rx 180 ry 0 rz 160 deg; joints [3.756, 78.749, -27.992, -150.39, 54.62, 161.786]
  Set speed (17.7 mm/s)
  Call Extruder(636.87214)
  MoveL 3766 to (560.01, 485.74, 64) mm, rotated rx 180 ry 0 rz 160 deg; joints [3.898, 78.838, -28.177, -150.191, 54.581, 161.632]
  Call Extruder(640.79243)
  MoveL 3767 to (560.29, 486.94, 64) mm, rotated rx -180 ry 0 rz 160 deg; joints [4.029, 78.919, -28.345, -150.007, 54.547, 161.49]
  Set speed (17.7 mm/s)
  Call Extruder(648.92429)
  MoveL 3768 to (560.77, 489.44, 64) mm, rotated rx -180 ry 0 rz 160 deg; joints [4.305, 79.07, -28.657, -149.629, 54.495, 161.204]
  Set speed (17.7 mm/s)
  Call Extruder(656.90751)
  MoveL 3769 to (561.15, 491.91, 64) mm, rotated rx 180 ry 0 rz 160 deg; joints [4.578, 79.199, -28.925, -149.261, 54.464, 160.933]
  Set speed (17.7 mm/s)
  Call Extruder(665.12638)
  MoveL 3770 to (561.44, 494.47, 64) mm, rotated rx 180 ry 0 rz 160 deg; joints [4.86, 79.311, -29.158, -148.889, 54.454, 160.666]
  Set speed (17.7 mm/s)
  Call Extruder(673.07383)
  MoveL 3771 to (561.61, 496.96, 64) mm, rotated rx 180 ry 0 rz 160 deg; joints [5.135, 79.401, -29.343, -148.535, 54.463, 160.42]
  Set speed (17.7 mm/s)
  Call Extruder(681.12618)
  MoveL 3772 to (561.68, 499.48, 64) mm, rotated rx 180 ry 0 rz 160 deg; joints [5.415, 79.47, -29.488, -148.183, 54.494, 160.184]
  Set speed (17.7 mm/s)
  Call Extruder(689.26360)
  MoveL 3773 to (561.65, 502.03, 64) mm, rotated rx -180 ry 0 rz 160 deg; joints [5.699, 79.52, -29.591, -147.835, 54.545, 159.959]
  Set speed (17.7 mm/s)
  Call Extruder(697.22843)
  MoveL 3774 to (561.52, 504.53, 64) mm, rotated rx 180 ry 0 rz 160 deg; joints [5.977, 79.548, -29.648, -147.503, 54.616, 159.754]
  Call Extruder(705.18755)
  MoveL 3775 to (561.29, 507.01, 64) mm, rotated rx -180 ry 0 rz 160 deg; joints [6.256, 79.556, -29.664, -147.18, 54.706, 159.563]
  Set speed (17.7 mm/s)
  Call Extruder(713.41822)
  MoveL 3776 to (560.94, 509.57, 64) mm, rotated rx -180 ry 0 rz 160 deg; joints [6.543, 79.542, -29.636, -146.856, 54.819, 159.383]
  Call Extruder(721.36449)
  MoveL 3777 to (560.5, 512.02, 64) mm, rotated rx 180 ry 0 rz 160 deg; joints [6.821, 79.508, -29.566, -146.553, 54.947, 159.224]
  Call Extruder(729.47185)
  MoveL 3778 to (559.96, 514.5, 64) mm, rotated rx -180 ry 0 rz 160 deg; joints [7.103, 79.452, -29.45, -146.254, 55.098, 159.08]
  Set speed (17.7 mm/s)
  Call Extruder(733.47851)
  MoveL 3779 to (559.64, 515.72, 64) mm, rotated rx -180 ry 0 rz 160 deg; joints [7.242, 79.416, -29.375, -146.111, 55.18, 159.016]
  Set speed (17.7 mm/s)
  Call Extruder(737.39895)
  MoveL 3780 to (559.33, 516.9, 64) mm, rotated rx -180 ry 0 rz 160 deg; joints [7.378, 79.378, -29.296, -145.972, 55.262, 158.956]
  Set speed (17.7 mm/s)
  Call Extruder(741.54282)
  MoveL 3781 to (558.95, 518.14, 64) mm, rotated rx 180 ry 0 rz 160 deg; joints [7.521, 79.329, -29.196, -145.83, 55.357, 158.899]
  Call Extruder(745.62914)
  MoveL 3782 to (558.57, 519.36, 64) mm, rotated rx -180 ry 0 rz 160 deg; joints [7.662, 79.28, -29.093, -145.691, 55.452, 158.844]
  Set speed (17.7 mm/s)
  Call Extruder(753.74348)
  MoveL 3783 to (557.72, 521.76, 64) mm, rotated rx -180 ry 0 rz 160 deg; joints [7.941, 79.163, -28.85, -145.424, 55.656, 158.752]
  Set speed (17.7 mm/s)
  Call Extruder(761.58721)
  MoveL 3784 to (556.81, 524.05, 64) mm, rotated rx 180 ry 0 rz 160 deg; joints [8.208, 79.031, -28.576, -145.178, 55.87, 158.68]
  Set speed (17.7 mm/s)
  Call Extruder(769.51855)
  MoveL 3785 to (555.79, 526.32, 64) mm, rotated rx -180 ry 0 rz 160 deg; joints [8.477, 78.879, -28.261, -144.94, 56.102, 158.625]
  Set speed (17.7 mm/s)
  Call Extruder(773.77616)
  MoveL 3786 to (555.21, 527.52, 64) mm, rotated rx 180 ry 0 rz 160 deg; joints [8.62, 78.79, -28.075, -144.816, 56.233, 158.602]
  Set speed (17.7 mm/s)
  Call Extruder(777.65060)
  MoveL 3787 to (554.66, 528.6, 64) mm, rotated rx -180 ry 0 rz 160 deg; joints [8.749, 78.705, -27.899, -144.707, 56.355, 158.585]
  Set speed (17.7 mm/s)
  Call Extruder(781.68345)
  MoveL 3788 to (554.06, 529.71, 64) mm, rotated rx -180 ry 0 rz 160 deg; joints [8.883, 78.612, -27.705, -144.596, 56.486, 158.572]
  Set speed (17.7 mm/s)
  Call Extruder(785.07759)
  MoveL 3789 to (553.54, 530.64, 64) mm, rotated rx 180 ry 0 rz 160 deg; joints [8.996, 78.53, -27.534, -144.504, 56.599, 158.565]
  Set speed (17.7 mm/s)
  Call Extruder(789.70488)
  MoveL 3790 to (552.8, 531.89, 64) mm, rotated rx 180 ry 0 rz 160 deg; joints [9.148, 78.414, -27.293, -144.383, 56.757, 158.559]
  Call Extruder(793.80517)
  MoveL 3791 to (552.13, 532.99, 64) mm, rotated rx -180 ry 0 rz 160 deg; joints [9.282, 78.306, -27.069, -144.278, 56.901, 158.559]
  Set speed (17.7 mm/s)
  Call Extruder(797.80222)
  MoveL 3792 to (551.44, 534.04, 64) mm, rotated rx -180 ry 0 rz 160 deg; joints [9.411, 78.197, -26.841, -144.18, 57.044, 158.563]
  Set speed (17.7 mm/s)
  Call Extruder(802.01389)
  MoveL 3793 to (550.71, 535.13, 64) mm, rotated rx -180 ry 0 rz 160 deg; joints [9.547, 78.078, -26.593, -144.078, 57.198, 158.572]
  Set speed (17.7 mm/s)
  Call Extruder(805.82527)
  MoveL 3794 to (550.01, 536.11, 64) mm, rotated rx -180 ry 0 rz 160 deg; joints [9.668, 77.967, -26.36, -143.989, 57.341, 158.584]
  Call Extruder(809.91421)
  MoveL 3795 to (549.25, 537.14, 64) mm, rotated rx 180 ry 0 rz 160 deg; joints [9.798, 77.843, -26.102, -143.897, 57.497, 158.601]
  Call Extruder(813.95993)
  MoveL 3796 to (548.48, 538.14, 64) mm, rotated rx -180 ry 0 rz 160 deg; joints [9.925, 77.718, -25.84, -143.808, 57.654, 158.621]
  Set speed (17.7 mm/s)
  Call Extruder(817.98520)
  MoveL 3797 to (547.69, 539.12, 64) mm, rotated rx -180 ry 0 rz 160 deg; joints [10.051, 77.589, -25.57, -143.722, 57.813, 158.646]
  Call Extruder(821.93922)
  MoveL 3798 to (546.89, 540.08, 64) mm, rotated rx -180 ry 0 rz 160 deg; joints [10.173, 77.459, -25.298, -143.641, 57.972, 158.674]
  Call Extruder(825.96167)
  MoveL 3799 to (546.07, 541.02, 64) mm, rotated rx -180 ry 0 rz 160 deg; joints [10.296, 77.324, -25.014, -143.561, 58.137, 158.706]
  Set speed (17.7 mm/s)
  Call Extruder(830.10442)
  MoveL 3800 to (545.19, 541.99, 64) mm, rotated rx 180 ry 0 rz 160 deg; joints [10.421, 77.181, -24.714, -143.481, 58.308, 158.743]
  Call Extruder(834.01141)
  MoveL 3801 to (544.35, 542.88, 64) mm, rotated rx -180 ry 0 rz 160 deg; joints [10.539, 77.043, -24.425, -143.408, 58.473, 158.782]
  Set speed (17.7 mm/s)
  Call Extruder(838.04654)
  MoveL 3802 to (543.46, 543.77, 64) mm, rotated rx -180 ry 0 rz 160 deg; joints [10.658, 76.897, -24.119, -143.336, 58.644, 158.826]
  Set speed (17.7 mm/s)
  Call Extruder(842.08563)
  MoveL 3803 to (542.55, 544.66, 64) mm, rotated rx 180 ry 0 rz 160 deg; joints [10.777, 76.749, -23.807, -143.266, 58.818, 158.873]
  Set speed (17.7 mm/s)
  Call Extruder(846.96652)
  MoveL 3804 to (541.43, 545.7, 64) mm, rotated rx -180 ry 0 rz 160 deg; joints [10.918, 76.566, -23.422, -143.185, 59.031, 158.935]
  Set speed (17.7 mm/s)
  Call Extruder(850.12450)
  MoveL 3805 to (540.7, 546.36, 64) mm, rotated rx 180 ry 0 rz 160 deg; joints [11.008, 76.445, -23.166, -143.135, 59.171, 158.979]
  Set speed (17.7 mm/s)
  Call Extruder(854.26284)
  MoveL 3806 to (539.71, 547.2, 64) mm, rotated rx -180 ry 0 rz 160 deg; joints [11.125, 76.284, -22.827, -143.072, 59.356, 159.039]
  Call Extruder(858.22750)
  MoveL 3807 to (538.75, 547.99, 64) mm, rotated rx 180 ry 0 rz 160 deg; joints [11.236, 76.128, -22.497, -143.014, 59.534, 159.099]
  Set speed (17.7 mm/s)
  Call Extruder(862.19406)
  MoveL 3808 to (537.78, 548.77, 64) mm, rotated rx 180 ry 0 rz 160 deg; joints [11.345, 75.969, -22.161, -142.958, 59.714, 159.163]
  Set speed (17.7 mm/s)
  Call Extruder(866.21463)
  MoveL 3809 to (536.77, 549.52, 64) mm, rotated rx -180 ry 0 rz 160 deg; joints [11.454, 75.806, -21.815, -142.904, 59.899, 159.231]
  Set speed (17.7 mm/s)
  Call Extruder(870.29974)
  MoveL 3810 to (535.74, 550.28, 64) mm, rotated rx -180 ry 0 rz 160 deg; joints [11.563, 75.637, -21.458, -142.852, 60.088, 159.303]
  Set speed (17.7 mm/s)
  Call Extruder(874.27866)
  MoveL 3811 to (534.71, 550.99, 64) mm, rotated rx 180 ry 0 rz 160 deg; joints [11.668, 75.471, -21.105, -142.803, 60.273, 159.377]
  Call Extruder(878.34088)
  MoveL 3812 to (533.65, 551.7, 64) mm, rotated rx -180 ry 0 rz 160 deg; joints [11.773, 75.3, -20.741, -142.756, 60.464, 159.455]
  Set speed (17.7 mm/s)
  Call Extruder(882.32891)
  MoveL 3813 to (532.6, 552.37, 64) mm, rotated rx -180 ry 0 rz 160 deg; joints [11.875, 75.129, -20.379, -142.713, 60.652, 159.535]
  Set speed (17.7 mm/s)
  Call Extruder(886.38019)
  MoveL 3814 to (531.52, 553.03, 64) mm, rotated rx -180 ry 0 rz 160 deg; joints [11.976, 74.954, -20.007, -142.671, 60.844, 159.619]
  Set speed (17.7 mm/s)
  Call Extruder(890.41881)
  MoveL 3815 to (530.42, 553.66, 64) mm, rotated rx 180 ry 0 rz 160 deg; joints [12.075, 74.778, -19.631, -142.632, 61.038, 159.706]
  Set speed (17.7 mm/s)
  Call Extruder(894.39484)
  MoveL 3816 to (529.33, 554.27, 64) mm, rotated rx 180 ry 0 rz 160 deg; joints [12.171, 74.603, -19.257, -142.596, 61.229, 159.794]
  Set speed (17.7 mm/s)
  Call Extruder(898.42062)
  MoveL 3817 to (528.21, 554.86, 64) mm, rotated rx 180 ry 0 rz 160 deg; joints [12.266, 74.424, -18.875, -142.561, 61.423, 159.886]
  Set speed (17.7 mm/s)
  Call Extruder(902.44052)
  MoveL 3818 to (527.09, 555.42, 64) mm, rotated rx -180 ry 0 rz 160 deg; joints [12.359, 74.244, -18.489, -142.53, 61.617, 159.98]
  Set speed (17.7 mm/s)
  Call Extruder(906.60995)
  MoveL 3819 to (525.91, 555.99, 64) mm, rotated rx -180 ry 0 rz 160 deg; joints [12.453, 74.056, -18.088, -142.499, 61.82, 160.08]
  Set speed (17.7 mm/s)
  Call Extruder(910.57814)
  MoveL 3820 to (524.77, 556.49, 64) mm, rotated rx -180 ry 0 rz 160 deg; joints [12.54, 73.875, -17.7, -142.474, 62.014, 160.18]
  Set speed (17.7 mm/s)
  Call Extruder(914.52413)
  MoveL 3821 to (523.64, 556.98, 64) mm, rotated rx 180 ry 0 rz 160 deg; joints [12.626, 73.696, -17.314, -142.449, 62.206, 160.279]
  Set speed (17.7 mm/s)
  Call Extruder(918.63866)
  MoveL 3822 to (522.44, 557.45, 64) mm, rotated rx 180 ry 0 rz 160 deg; joints [12.712, 73.506, -16.906, -142.428, 62.408, 160.387]
  Call Extruder(922.73096)
  MoveL 3823 to (521.25, 557.91, 64) mm, rotated rx 180 ry 0 rz 160 deg; joints [12.796, 73.318, -16.501, -142.407, 62.608, 160.495]
  Set speed (17.7 mm/s)
  Call Extruder(930.60506)
  MoveL 3824 to (518.91, 558.72, 64) mm, rotated rx 180 ry 0 rz 160 deg; joints [12.951, 72.952, -15.711, -142.375, 62.996, 160.711]
  Set speed (17.7 mm/s)
  Call Extruder(934.74946)
  MoveL 3825 to (517.67, 559.09, 64) mm, rotated rx -180 ry 0 rz 160 deg; joints [13.029, 72.757, -15.29, -142.364, 63.2, 160.829]
  Set speed (17.7 mm/s)
  Call Extruder(938.63456)
  MoveL 3826 to (516.51, 559.44, 64) mm, rotated rx -180 ry 0 rz 160 deg; joints [13.1, 72.576, -14.896, -142.353, 63.391, 160.939]
  Set speed (17.7 mm/s)
  Call Extruder(942.27803)
  MoveL 3827 to (515.4, 559.73, 64) mm, rotated rx 180 ry 0 rz 160 deg; joints [13.164, 72.404, -14.524, -142.347, 63.571, 161.046]
  Set speed (17.7 mm/s)
  Call Extruder(946.72258)
  MoveL 3828 to (514.05, 560.06, 64) mm, rotated rx 180 ry 0 rz 160 deg; joints [13.241, 72.195, -14.07, -142.34, 63.79, 161.178]
  Set speed (17.7 mm/s)
  Call Extruder(954.89726)
  MoveL 3829 to (511.55, 560.6, 64) mm, rotated rx -180 ry 0 rz 160 deg; joints [13.373, 71.808, -13.227, -142.336, 64.193, 161.426]
  Set speed (17.7 mm/s)
  Call Extruder(963.00256)
  MoveL 3830 to (509.04, 561.02, 64) mm, rotated rx -180 ry 0 rz 160 deg; joints [13.493, 71.423, -12.387, -142.343, 64.592, 161.68]
  Set speed (17.7 mm/s)
  Call Extruder(970.98119)
  MoveL 3831 to (506.56, 561.34, 64) mm, rotated rx 180 ry 0 rz 160 deg; joints [13.601, 71.044, -11.556, -142.359, 64.983, 161.937]
  Call Extruder(979.07957)
  MoveL 3832 to (504.03, 561.55, 64) mm, rotated rx -180 ry 0 rz 160 deg; joints [13.701, 70.66, -10.711, -142.385, 65.379, 162.203]
  Set speed (17.7 mm/s)
  Call Extruder(987.17189)
  MoveL 3833 to (501.5, 561.67, 64) mm, rotated rx 180 ry 0 rz 160 deg; joints [13.788, 70.277, -9.867, -142.422, 65.771, 162.474]
  Set speed (17.7 mm/s)
  Call Extruder(995.13331)
  MoveL 3834 to (499, 561.68, 64) mm, rotated rx -180 ry 0 rz 160 deg; joints [13.863, 69.902, -9.036, -142.467, 66.155, 162.746]
  Set speed (10.0 mm/s)
  MoveL 3835 to (499, 561.68, 68) mm, rotated rx 180 ry 0 rz 160 deg; joints [13.863, 69.226, -8.638, -142.392, 65.934, 162.561]
  Set speed (120.0 mm/s)
  MoveL 3836 to (499.02, 562.42, 68) mm, rotated rx 180 ry 0 rz 160 deg; joints [13.952, 69.256, -8.704, -142.289, 65.932, 162.499]
  Set speed (17.7 mm/s)
  Call Extruder(1003.41755)
  MoveL 3837 to (496.42, 562.32, 68) mm, rotated rx -180 ry 0 rz 160 deg; joints [14.018, 68.866, -7.843, -142.348, 66.325, 162.786]
  Set speed (17.7 mm/s)
  Call Extruder(1011.58774)
  MoveL 3838 to (493.86, 562.12, 68) mm, rotated rx 180 ry 0 rz 160 deg; joints [14.072, 68.484, -6.997, -142.415, 66.709, 163.073]
  Call Extruder(1019.64084)
  MoveL 3839 to (491.35, 561.82, 68) mm, rotated rx 180 ry 0 rz 160 deg; joints [14.112, 68.111, -6.166, -142.492, 67.083, 163.359]
  Set speed (17.7 mm/s)
  Call Extruder(1027.69677)
  MoveL 3840 to (488.86, 561.42, 68) mm, rotated rx 180 ry 0 rz 160 deg; joints [14.14, 67.741, -5.341, -142.579, 67.453, 163.649]
  Set speed (17.7 mm/s)
  Call Extruder(1036.00940)
  MoveL 3841 to (486.3, 560.9, 68) mm, rotated rx 180 ry 0 rz 160 deg; joints [14.156, 67.364, -4.495, -142.68, 67.829, 163.95]
  Set speed (17.7 mm/s)
  Call Extruder(1040.02611)
  MoveL 3842 to (485.08, 560.61, 68) mm, rotated rx 180 ry 0 rz 160 deg; joints [14.157, 67.184, -4.09, -142.733, 68.008, 164.096]
  Set speed (17.7 mm/s)
  Call Extruder(1043.93126)
  MoveL 3843 to (483.89, 560.31, 68) mm, rotated rx -180 ry 0 rz 160 deg; joints [14.157, 67.01, -3.699, -142.787, 68.182, 164.239]
  Call Extruder(1048.11762)
  MoveL 3844 to (482.62, 559.95, 68) mm, rotated rx -180 ry 0 rz 160 deg; joints [14.152, 66.825, -3.281, -142.848, 68.366, 164.392]
  Set speed (17.7 mm/s)
  Call Extruder(1052.13919)
  MoveL 3845 to (481.42, 559.59, 68) mm, rotated rx -180 ry 0 rz 160 deg; joints [14.146, 66.648, -2.881, -142.907, 68.542, 164.539]
  Call Extruder(1056.27531)
  MoveL 3846 to (480.18, 559.19, 68) mm, rotated rx 180 ry 0 rz 160 deg; joints [14.134, 66.468, -2.474, -142.973, 68.72, 164.691]
  Set speed (17.7 mm/s)
  Call Extruder(1060.25936)
  MoveL 3847 to (479, 558.79, 68) mm, rotated rx 180 ry 0 rz 160 deg; joints [14.121, 66.296, -2.083, -143.038, 68.891, 164.837]
  Set speed (17.7 mm/s)
  Call Extruder(1064.44419)
  MoveL 3848 to (477.77, 558.33, 68) mm, rotated rx -180 ry 0 rz 160 deg; joints [14.102, 66.117, -1.676, -143.11, 69.069, 164.991]
  Call Extruder(1068.67923)
  MoveL 3849 to (476.53, 557.85, 68) mm, rotated rx -180 ry 0 rz 160 deg; joints [14.081, 65.937, -1.266, -143.185, 69.247, 165.146]
  Call Extruder(1075.50468)
  MoveL 3850 to (474.57, 557.01, 68) mm, rotated rx -180 ry 0 rz 160 deg; joints [14.037, 65.651, -0.613, -143.313, 69.531, 165.397]
  Set speed (17.7 mm/s)
  Call Extruder(1080.65798)
  MoveL 3851 to (473.1, 556.33, 68) mm, rotated rx -180 ry 0 rz 160 deg; joints [13.997, 65.439, -0.125, -143.414, 69.741, 165.586]
  Set speed (17.7 mm/s)
  Call Extruder(1084.77852)
  MoveL 3852 to (471.94, 555.76, 68) mm, rotated rx 180 ry 0 rz 160 deg; joints [13.961, 65.271, 0.261, -143.499, 69.907, 165.737]
  Set speed (17.7 mm/s)
  Call Extruder(1088.79181)
  MoveL 3853 to (470.82, 555.18, 68) mm, rotated rx 180 ry 0 rz 160 deg; joints [13.923, 65.109, 0.633, -143.585, 70.067, 165.884]
  Set speed (17.7 mm/s)
  Call Extruder(1092.81523)
  MoveL 3854 to (469.71, 554.58, 68) mm, rotated rx -180 ry 0 rz 160 deg; joints [13.881, 64.948, 1.003, -143.673, 70.226, 166.03]
  Call Extruder(1097.07343)
  MoveL 3855 to (468.55, 553.92, 68) mm, rotated rx 180 ry 0 rz 160 deg; joints [13.832, 64.78, 1.391, -143.769, 70.392, 166.185]
  Call Extruder(1101.62493)
  MoveL 3856 to (467.32, 553.19, 68) mm, rotated rx -180 ry 0 rz 160 deg; joints [13.776, 64.603, 1.801, -143.876, 70.566, 166.351]
  Call Extruder(1105.10597)
  MoveL 3857 to (466.39, 552.61, 68) mm, rotated rx -180 ry 0 rz 160 deg; joints [13.73, 64.47, 2.111, -143.96, 70.698, 166.476]
  Set speed (17.7 mm/s)
  Call Extruder(1109.12586)
  MoveL 3858 to (465.34, 551.91, 68) mm, rotated rx 180 ry 0 rz 160 deg; joints [13.674, 64.317, 2.465, -144.059, 70.848, 166.621]
  Set speed (17.7 mm/s)
  Call Extruder(1113.20597)
  MoveL 3859 to (464.28, 551.19, 68) mm, rotated rx 180 ry 0 rz 160 deg; joints [13.613, 64.165, 2.821, -144.163, 70.998, 166.768]
  Set speed (17.7 mm/s)
  Call Extruder(1117.23122)
  MoveL 3860 to (463.25, 550.46, 68) mm, rotated rx 180 ry 0 rz 160 deg; joints [13.549, 64.016, 3.167, -144.268, 71.145, 166.911]
  Set speed (17.7 mm/s)
  Call Extruder(1121.41242)
  MoveL 3861 to (462.2, 549.68, 68) mm, rotated rx 180 ry 0 rz 160 deg; joints [13.48, 63.864, 3.523, -144.38, 71.294, 167.06]
  Set speed (17.7 mm/s)
  Call Extruder(1125.34561)
  MoveL 3862 to (461.22, 548.92, 68) mm, rotated rx 180 ry 0 rz 160 deg; joints [13.41, 63.724, 3.852, -144.488, 71.432, 167.198]
  Set speed (17.7 mm/s)
  Call Extruder(1129.45251)
  MoveL 3863 to (460.22, 548.11, 68) mm, rotated rx 180 ry 0 rz 160 deg; joints [13.335, 63.579, 4.192, -144.604, 71.575, 167.342]
  Call Extruder(1133.53297)
  MoveL 3864 to (459.24, 547.28, 68) mm, rotated rx -180 ry 0 rz 160 deg; joints [13.256, 63.438, 4.524, -144.722, 71.713, 167.484]
  Set speed (17.7 mm/s)
  Call Extruder(1137.54951)
  MoveL 3865 to (458.29, 546.45, 68) mm, rotated rx 180 ry 0 rz 160 deg; joints [13.174, 63.301, 4.847, -144.841, 71.848, 167.623]
  Set speed (17.7 mm/s)
  Call Extruder(1141.67068)
  MoveL 3866 to (457.34, 545.57, 68) mm, rotated rx 180 ry 0 rz 160 deg; joints [13.087, 63.163, 5.173, -144.966, 71.983, 167.765]
  Call Extruder(1145.72595)
  MoveL 3867 to (456.42, 544.69, 68) mm, rotated rx 180 ry 0 rz 160 deg; joints [12.998, 63.03, 5.488, -145.091, 72.113, 167.903]
  Set speed (17.7 mm/s)
  Call Extruder(1149.76966)
  MoveL 3868 to (455.52, 543.8, 68) mm, rotated rx -180 ry 0 rz 160 deg; joints [12.906, 62.899, 5.798, -145.219, 72.241, 168.039]
  Call Extruder(1153.86368)
  MoveL 3869 to (454.63, 542.87, 68) mm, rotated rx 180 ry 0 rz 160 deg; joints [12.808, 62.77, 6.105, -145.351, 72.367, 168.176]
  Set speed (17.7 mm/s)
  Call Extruder(1158.74328)
  MoveL 3870 to (453.59, 541.75, 68) mm, rotated rx -180 ry 0 rz 160 deg; joints [12.688, 62.619, 6.465, -145.512, 72.515, 168.337]
  Set speed (17.7 mm/s)
  Call Extruder(1161.93740)
  MoveL 3871 to (452.93, 540.99, 68) mm, rotated rx -180 ry 0 rz 160 deg; joints [12.606, 62.522, 6.695, -145.62, 72.609, 168.442]
  Set speed (17.7 mm/s)
  Call Extruder(1165.62777)
  MoveL 3872 to (452.17, 540.11, 68) mm, rotated rx -180 ry 0 rz 160 deg; joints [12.51, 62.412, 6.959, -145.746, 72.716, 168.562]
  Set speed (17.7 mm/s)
  Call Extruder(1170.18065)
  MoveL 3873 to (451.26, 539.01, 68) mm, rotated rx 180 ry 0 rz 160 deg; joints [12.386, 62.279, 7.276, -145.905, 72.844, 168.708]
  Set speed (17.7 mm/s)
  Call Extruder(1174.20961)
  MoveL 3874 to (450.49, 538.01, 68) mm, rotated rx -180 ry 0 rz 160 deg; joints [12.273, 62.165, 7.55, -146.048, 72.955, 168.836]
  Call Extruder(1178.26652)
  MoveL 3875 to (449.72, 536.99, 68) mm, rotated rx -180 ry 0 rz 160 deg; joints [12.157, 62.053, 7.821, -146.195, 73.064, 168.963]
  Set speed (17.7 mm/s)
  Call Extruder(1182.31888)
  MoveL 3876 to (448.98, 535.96, 68) mm, rotated rx 180 ry 0 rz 160 deg; joints [12.037, 61.943, 8.085, -146.344, 73.169, 169.088]
  Set speed (17.7 mm/s)
  Call Extruder(1186.48230)
  MoveL 3877 to (448.23, 534.89, 68) mm, rotated rx 180 ry 0 rz 160 deg; joints [11.91, 61.833, 8.351, -146.5, 73.275, 169.216]
  Set speed (17.7 mm/s)
  Call Extruder(1190.48070)
  MoveL 3878 to (447.54, 533.84, 68) mm, rotated rx 180 ry 0 rz 160 deg; joints [11.785, 61.73, 8.599, -146.652, 73.373, 169.336]
  Call Extruder(1194.51902)
  MoveL 3879 to (446.87, 532.77, 68) mm, rotated rx 180 ry 0 rz 160 deg; joints [11.656, 61.629, 8.844, -146.808, 73.47, 169.456]
  Set speed (17.7 mm/s)
  Call Extruder(1198.55186)
  MoveL 3880 to (446.21, 531.68, 68) mm, rotated rx 180 ry 0 rz 160 deg; joints [11.524, 61.531, 9.082, -146.966, 73.563, 169.574]
  Call Extruder(1201.96590)
  MoveL 3881 to (445.68, 530.75, 68) mm, rotated rx -180 ry 0 rz 160 deg; joints [11.41, 61.45, 9.278, -147.101, 73.639, 169.673]
  Set speed (17.7 mm/s)
  Call Extruder(1206.11714)
  MoveL 3882 to (445.05, 529.61, 68) mm, rotated rx -180 ry 0 rz 160 deg; joints [11.269, 61.355, 9.51, -147.268, 73.729, 169.791]
  Call Extruder(1210.73332)
  MoveL 3883 to (444.37, 528.33, 68) mm, rotated rx 180 ry 0 rz 160 deg; joints [11.108, 61.252, 9.761, -147.456, 73.825, 169.92]
  Set speed (17.7 mm/s)
  Call Extruder(1216.00887)
  MoveL 3884 to (443.64, 526.85, 68) mm, rotated rx -180 ry 0 rz 160 deg; joints [10.919, 61.139, 10.035, -147.675, 73.929, 170.064]
  Call Extruder(1223.02717)
  MoveL 3885 to (442.73, 524.84, 68) mm, rotated rx 180 ry 0 rz 160 deg; joints [10.662, 60.997, 10.384, -147.97, 74.059, 170.251]
  Set speed (17.7 mm/s)
  Call Extruder(1227.16414)
  MoveL 3886 to (442.23, 523.65, 68) mm, rotated rx 180 ry 0 rz 160 deg; joints [10.506, 60.918, 10.577, -148.147, 74.13, 170.358]
  Call Extruder(1231.05438)
  MoveL 3887 to (441.78, 522.51, 68) mm, rotated rx 180 ry 0 rz 160 deg; joints [10.357, 60.846, 10.755, -148.315, 74.195, 170.457]
  Call Extruder(1235.31512)
  MoveL 3888 to (441.32, 521.26, 68) mm, rotated rx -180 ry 0 rz 160 deg; joints [10.191, 60.771, 10.94, -148.501, 74.261, 170.563]
  Set speed (17.7 mm/s)
  Call Extruder(1239.38562)
  MoveL 3889 to (440.89, 520.06, 68) mm, rotated rx -180 ry 0 rz 160 deg; joints [10.031, 60.701, 11.112, -148.68, 74.322, 170.663]
  Set speed (17.7 mm/s)
  Call Extruder(1247.52682)
  MoveL 3890 to (440.11, 517.62, 68) mm, rotated rx 180 ry 0 rz 160 deg; joints [9.703, 60.571, 11.431, -149.044, 74.432, 170.855]
  Set speed (17.7 mm/s)
  Call Extruder(1251.60119)
  MoveL 3891 to (439.77, 516.39, 68) mm, rotated rx 180 ry 0 rz 160 deg; joints [9.535, 60.512, 11.578, -149.229, 74.481, 170.948]
  Set speed (17.7 mm/s)
  Call Extruder(1255.52076)
  MoveL 3892 to (439.46, 515.21, 68) mm, rotated rx 180 ry 0 rz 160 deg; joints [9.372, 60.457, 11.715, -149.407, 74.525, 171.036]
  Set speed (17.7 mm/s)
  Call Extruder(1259.72729)
  MoveL 3893 to (439.15, 513.92, 68) mm, rotated rx 180 ry 0 rz 160 deg; joints [9.195, 60.402, 11.851, -149.6, 74.568, 171.127]
  Set speed (17.7 mm/s)
  Call Extruder(1263.77602)
  MoveL 3894 to (438.88, 512.68, 68) mm, rotated rx -180 ry 0 rz 160 deg; joints [9.023, 60.351, 11.977, -149.787, 74.607, 171.213]
  Set speed (17.7 mm/s)
  Call Extruder(1271.97143)
  MoveL 3895 to (438.41, 510.15, 68) mm, rotated rx 180 ry 0 rz 160 deg; joints [8.669, 60.259, 12.206, -150.169, 74.671, 171.38]
  Set speed (17.7 mm/s)
  Call Extruder(1280.11292)
  MoveL 3896 to (438.04, 507.62, 68) mm, rotated rx -180 ry 0 rz 160 deg; joints [8.311, 60.179, 12.404, -150.552, 74.721, 171.538]
  Set speed (17.7 mm/s)
  Call Extruder(1288.23087)
  MoveL 3897 to (437.79, 505.09, 68) mm, rotated rx -180 ry 0 rz 160 deg; joints [7.949, 60.113, 12.568, -150.936, 74.754, 171.685]
  Set speed (17.7 mm/s)
  Call Extruder(1296.22155)
  MoveL 3898 to (437.63, 502.59, 68) mm, rotated rx 180 ry 0 rz 160 deg; joints [7.588, 60.061, 12.699, -151.317, 74.771, 171.822]
  Set speed (17.7 mm/s)
  Call Extruder(1304.43193)
  MoveL 3899 to (437.58, 500.01, 68) mm, rotated rx 180 ry 0 rz 160 deg; joints [7.214, 60.019, 12.802, -151.708, 74.773, 171.953]
  Set speed (17.7 mm/s)
  Call Extruder(1311.82930)
  MoveL 3900 to (437.62, 497.69, 68) mm, rotated rx -180 ry 0 rz 160 deg; joints [6.875, 59.993, 12.867, -152.062, 74.76, 172.064]
  Call Extruder(1319.01371)
  MoveL 3901 to (437.74, 495.44, 68) mm, rotated rx 180 ry 0 rz 160 deg; joints [6.544, 59.979, 12.904, -152.405, 74.734, 172.164]
  Set speed (17.7 mm/s)
  Call Extruder(1326.39596)
  MoveL 3902 to (437.96, 493.13, 68) mm, rotated rx -180 ry 0 rz 160 deg; joints [6.203, 59.974, 12.916, -152.755, 74.694, 172.26]
  Set speed (17.7 mm/s)
  Call Extruder(1333.71516)
  MoveL 3903 to (438.25, 490.85, 68) mm, rotated rx -180 ry 0 rz 160 deg; joints [5.865, 59.98, 12.902, -153.101, 74.641, 172.347]
  Set speed (17.7 mm/s)
  Call Extruder(1340.86862)
  MoveL 3904 to (438.62, 488.64, 68) mm, rotated rx -180 ry 0 rz 160 deg; joints [5.536, 59.995, 12.863, -153.437, 74.577, 172.426]
  Set speed (17.7 mm/s)
  Call Extruder(1348.30177)
  MoveL 3905 to (439.09, 486.35, 68) mm, rotated rx 180 ry 0 rz 160 deg; joints [5.195, 60.022, 12.795, -153.783, 74.496, 172.501]
  Set speed (17.7 mm/s)
  Call Extruder(1355.73293)
  MoveL 3906 to (439.64, 484.09, 68) mm, rotated rx 180 ry 0 rz 160 deg; joints [4.856, 60.06, 12.702, -154.125, 74.402, 172.569]
  Call Extruder(1362.90632)
  MoveL 3907 to (440.25, 481.92, 68) mm, rotated rx -180 ry 0 rz 160 deg; joints [4.532, 60.106, 12.586, -154.45, 74.297, 172.628]
  Call Extruder(1370.24403)
  MoveL 3908 to (440.96, 479.73, 68) mm, rotated rx -180 ry 0 rz 160 deg; joints [4.204, 60.164, 12.442, -154.778, 74.177, 172.681]
  Set speed (17.7 mm/s)
  Call Extruder(1377.72203)
  MoveL 3909 to (441.77, 477.52, 68) mm, rotated rx -180 ry 0 rz 160 deg; joints [3.874, 60.234, 12.268, -155.105, 74.041, 172.729]
  Set speed (17.7 mm/s)
  Call Extruder(1385.04624)
  MoveL 3910 to (442.63, 475.39, 68) mm, rotated rx 180 ry 0 rz 160 deg; joints [3.555, 60.312, 12.073, -155.42, 73.895, 172.769]
  Call Extruder(1392.36220)
  MoveL 3911 to (443.58, 473.3, 68) mm, rotated rx 180 ry 0 rz 160 deg; joints [3.242, 60.401, 11.852, -155.728, 73.736, 172.802]
  Set speed (17.7 mm/s)
  Call Extruder(1399.53026)
  MoveL 3912 to (444.58, 471.28, 68) mm, rotated rx 180 ry 0 rz 160 deg; joints [2.942, 60.498, 11.612, -156.021, 73.567, 172.829]
  Set speed (17.7 mm/s)
  Call Extruder(1406.91875)
  MoveL 3913 to (445.68, 469.24, 68) mm, rotated rx 180 ry 0 rz 160 deg; joints [2.638, 60.608, 11.341, -156.316, 73.382, 172.85]
  Call Extruder(1414.32977)
  MoveL 3914 to (446.86, 467.24, 68) mm, rotated rx -180 ry 0 rz 160 deg; joints [2.341, 60.728, 11.044, -156.603, 73.183, 172.865]
  Set speed (17.7 mm/s)
  Call Extruder(1421.55297)
  MoveL 3915 to (448.09, 465.33, 68) mm, rotated rx -180 ry 0 rz 160 deg; joints [2.059, 60.855, 10.731, -156.873, 72.977, 172.873]
  Set speed (17.7 mm/s)
  Call Extruder(1428.78110)
  MoveL 3916 to (449.38, 463.47, 68) mm, rotated rx 180 ry 0 rz 160 deg; joints [1.785, 60.992, 10.395, -157.134, 72.76, 172.876]
  Set speed (17.7 mm/s)
  Call Extruder(1436.19218)
  MoveL 3917 to (450.78, 461.6, 68) mm, rotated rx -180 ry 0 rz 160 deg; joints [1.512, 61.143, 10.027, -157.391, 72.526, 172.872]
  Set speed (17.7 mm/s)
  Call Extruder(1443.59349)
  MoveL 3918 to (452.25, 459.8, 68) mm, rotated rx 180 ry 0 rz 160 deg; joints [1.249, 61.303, 9.637, -157.637, 72.28, 172.862]
  Set speed (17.7 mm/s)
  Call Extruder(1450.82660)
  MoveL 3919 to (453.74, 458.09, 68) mm, rotated rx -180 ry 0 rz 160 deg; joints [1.002, 61.468, 9.234, -157.866, 72.03, 172.847]
  Set speed (17.7 mm/s)
  Call Extruder(1458.23213)
  MoveL 3920 to (455.33, 456.39, 68) mm, rotated rx -180 ry 0 rz 160 deg; joints [0.758, 61.647, 8.8, -158.089, 71.763, 172.826]
  Set speed (17.7 mm/s)
  Call Extruder(1465.42087)
  MoveL 3921 to (456.94, 454.81, 68) mm, rotated rx 180 ry 0 rz 160 deg; joints [0.531, 61.83, 8.358, -158.294, 71.494, 172.799]
  Set speed (17.7 mm/s)
  Call Extruder(1472.82888)
  MoveL 3922 to (458.65, 453.24, 68) mm, rotated rx -180 ry 0 rz 160 deg; joints [0.308, 62.027, 7.882, -158.493, 71.206, 172.765]
  Set speed (17.7 mm/s)
  Call Extruder(1480.14077)
  MoveL 3923 to (460.4, 451.75, 68) mm, rotated rx 180 ry 0 rz 160 deg; joints [0.098, 62.231, 7.392, -158.677, 70.914, 172.726]
  Set speed (17.7 mm/s)
  Call Extruder(1487.86602)
  MoveL 3924 to (462.3, 450.25, 68) mm, rotated rx -180 ry 0 rz 160 deg; joints [-0.111, 62.456, 6.854, -158.857, 70.595, 172.678]
  Set speed (17.7 mm/s)
  Call Extruder(1494.34388)
  MoveL 3925 to (463.94, 449.04, 68) mm, rotated rx -180 ry 0 rz 160 deg; joints [-0.277, 62.651, 6.388, -158.998, 70.321, 172.634]
  Set speed (17.7 mm/s)
  Call Extruder(1501.97503)
  MoveL 3926 to (465.92, 447.7, 68) mm, rotated rx 180 ry 0 rz 160 deg; joints [-0.461, 62.89, 5.82, -159.149, 69.99, 172.574]
  Set speed (17.7 mm/s)
  Call Extruder(1509.48743)
  MoveL 3927 to (467.92, 446.45, 68) mm, rotated rx 180 ry 0 rz 160 deg; joints [-0.631, 63.134, 5.242, -159.285, 69.655, 172.51]
  Set speed (17.7 mm/s)
  Call Extruder(1516.80464)
  MoveL 3928 to (469.91, 445.31, 68) mm, rotated rx -180 ry 0 rz 160 deg; joints [-0.784, 63.379, 4.662, -159.403, 69.323, 172.441]
  Set speed (17.7 mm/s)
  Call Extruder(1524.98415)
  MoveL 3929 to (472.18, 444.12, 68) mm, rotated rx -180 ry 0 rz 160 deg; joints [-0.942, 63.663, 3.995, -159.519, 68.943, 172.357]
  Set speed (17.7 mm/s)
  Call Extruder(1525.82651)
  MoveL 3930 to (472.42, 444.01, 68) mm, rotated rx -180 ry 0 rz 160 deg; joints [-0.956, 63.693, 3.924, -159.529, 68.903, 172.347]
  Set speed (17.7 mm/s)
  Call Extruder(1531.42827)
  MoveL 3931 to (474.01, 443.25, 68) mm, rotated rx 180 ry 0 rz 160 deg; joints [-1.055, 63.893, 3.456, -159.598, 68.638, 172.284]
  Set speed (17.7 mm/s)
  Call Extruder(1538.78305)
  MoveL 3932 to (476.12, 442.32, 68) mm, rotated rx -180 ry 0 rz 160 deg; joints [-1.174, 64.162, 2.826, -159.675, 68.284, 172.196]
  Call Extruder(1545.92991)
  MoveL 3933 to (478.21, 441.5, 68) mm, rotated rx -180 ry 0 rz 160 deg; joints [-1.278, 64.431, 2.201, -159.737, 67.936, 172.104]
  Set speed (17.7 mm/s)
  Call Extruder(1553.42389)
  MoveL 3934 to (480.43, 440.72, 68) mm, rotated rx 180 ry 0 rz 160 deg; joints [-1.376, 64.72, 1.532, -159.787, 67.565, 172.001]
  Set speed (17.7 mm/s)
  Call Extruder(1560.68015)
  MoveL 3935 to (482.61, 440.05, 68) mm, rotated rx -180 ry 0 rz 160 deg; joints [-1.458, 65.005, 0.871, -159.822, 67.202, 171.896]
  Call Extruder(1568.06218)
  MoveL 3936 to (484.84, 439.44, 68) mm, rotated rx 180 ry 0 rz 160 deg; joints [-1.53, 65.303, 0.187, -159.843, 66.828, 171.781]
  Call Extruder(0.00000)
  Call Extruder(7.23516)
  MoveL 3937 to (487.06, 438.93, 68) mm, rotated rx 180 ry 0 rz 160 deg; joints [-1.59, 65.6, -0.494, -159.849, 66.459, 171.662]
  Set speed (17.7 mm/s)
  Call Extruder(14.48849)
  MoveL 3938 to (489.29, 438.5, 68) mm, rotated rx 180 ry 0 rz 160 deg; joints [-1.638, 65.903, -1.188, -159.842, 66.086, 171.536]
  Call Extruder(21.54658)
  MoveL 3939 to (491.48, 438.16, 68) mm, rotated rx 180 ry 0 rz 160 deg; joints [-1.674, 66.203, -1.872, -159.823, 65.72, 171.407]
  Set speed (17.7 mm/s)
  Call Extruder(29.24011)
  MoveL 3940 to (493.88, 437.88, 68) mm, rotated rx -180 ry 0 rz 160 deg; joints [-1.702, 66.536, -2.626, -159.786, 65.32, 171.259]
  Call Extruder(36.45782)
  MoveL 3941 to (496.14, 437.7, 68) mm, rotated rx 180 ry 0 rz 160 deg; joints [-1.716, 66.852, -3.343, -159.737, 64.943, 171.114]
  Set speed (17.7 mm/s)
  Call Extruder(43.93273)
  MoveL 3942 to (498.48, 437.6, 68) mm, rotated rx -180 ry 0 rz 160 deg; joints [-1.72, 67.185, -4.092, -159.674, 64.551, 170.956]
  Set speed (17.7 mm/s)
  Call Extruder(51.17475)
  MoveL 3943 to (500.76, 437.58, 68) mm, rotated rx 180 ry 0 rz 160 deg; joints [-1.713, 67.511, -4.825, -159.599, 64.171, 170.796]
  Set speed (17.7 mm/s)
  Call Extruder(58.55419)
  MoveL 3944 to (503.07, 437.65, 68) mm, rotated rx 180 ry 0 rz 160 deg; joints [-1.696, 67.847, -5.578, -159.508, 63.783, 170.625]
  Call Extruder(65.80341)
  MoveL 3945 to (505.35, 437.81, 68) mm, rotated rx -180 ry 0 rz 160 deg; joints [-1.668, 68.181, -6.322, -159.406, 63.403, 170.45]
  Set speed (17.7 mm/s)
  Call Extruder(73.20399)
  MoveL 3946 to (507.66, 438.05, 68) mm, rotated rx -180 ry 0 rz 160 deg; joints [-1.629, 68.524, -7.086, -159.288, 63.017, 170.265]
  Set speed (17.7 mm/s)
  Call Extruder(80.36501)
  MoveL 3947 to (509.88, 438.37, 68) mm, rotated rx 180 ry 0 rz 160 deg; joints [-1.582, 68.859, -7.828, -159.161, 62.644, 170.079]
  Set speed (17.7 mm/s)
  Call Extruder(87.83871)
  MoveL 3948 to (512.19, 438.78, 68) mm, rotated rx -180 ry 0 rz 160 deg; joints [-1.522, 69.211, -8.605, -159.016, 62.256, 169.877]
  Call Extruder(94.94720)
  MoveL 3949 to (514.37, 439.25, 68) mm, rotated rx -180 ry 0 rz 160 deg; joints [-1.456, 69.547, -9.346, -158.866, 61.891, 169.678]
  Set speed (17.7 mm/s)
  Call Extruder(102.31918)
  MoveL 3950 to (516.62, 439.83, 68) mm, rotated rx 180 ry 0 rz 160 deg; joints [-1.379, 69.897, -10.115, -158.697, 61.514, 169.465]
  Set speed (17.7 mm/s)
  Call Extruder(109.87439)
  MoveL 3951 to (518.89, 440.51, 68) mm, rotated rx -180 ry 0 rz 160 deg; joints [-1.289, 70.257, -10.903, -158.512, 61.132, 169.239]
  Set speed (17.7 mm/s)
  Call Extruder(116.91887)
  MoveL 3952 to (520.99, 441.21, 68) mm, rotated rx -180 ry 0 rz 160 deg; joints [-1.197, 70.593, -11.637, -158.327, 60.78, 169.021]
  Set speed (17.7 mm/s)
  Call Extruder(124.33883)
  MoveL 3953 to (523.17, 442.03, 68) mm, rotated rx 180 ry 0 rz 160 deg; joints [-1.092, 70.947, -12.408, -158.122, 60.413, 168.786]
  Set speed (17.7 mm/s)
  Call Extruder(131.73705)
  MoveL 3954 to (525.31, 442.94, 68) mm, rotated rx 180 ry 0 rz 160 deg; joints [-0.978, 71.299, -13.172, -157.905, 60.053, 168.544]
  Set speed (17.7 mm/s)
  Call Extruder(138.97490)
  MoveL 3955 to (527.37, 443.9, 68) mm, rotated rx 180 ry 0 rz 160 deg; joints [-0.859, 71.643, -13.917, -157.682, 59.705, 168.301]
  Set speed (17.7 mm/s)
  Call Extruder(146.37829)
  MoveL 3956 to (529.44, 444.96, 68) mm, rotated rx 180 ry 0 rz 160 deg; joints [-0.728, 71.993, -14.673, -157.442, 59.357, 168.046]
  Set speed (17.7 mm/s)
  Call Extruder(153.69604)
  MoveL 3957 to (531.45, 446.08, 68) mm, rotated rx -180 ry 0 rz 160 deg; joints [-0.592, 72.338, -15.416, -157.196, 59.018, 167.788]
  Set speed (17.7 mm/s)
  Call Extruder(160.92294)
  MoveL 3958 to (533.38, 447.25, 68) mm, rotated rx -180 ry 0 rz 160 deg; joints [-0.45, 72.676, -16.141, -156.942, 58.692, 167.527]
  Set speed (17.7 mm/s)
  Call Extruder(168.33325)
  MoveL 3959 to (535.33, 448.54, 68) mm, rotated rx 180 ry 0 rz 160 deg; joints [-0.297, 73.019, -16.877, -156.672, 58.364, 167.254]
  Call Extruder(175.56330)
  MoveL 3960 to (537.17, 449.85, 68) mm, rotated rx 180 ry 0 rz 160 deg; joints [-0.14, 73.351, -17.587, -156.399, 58.053, 166.983]
  Set speed (17.7 mm/s)
  Call Extruder(182.91595)
  MoveL 3961 to (539, 451.26, 68) mm, rotated rx -180 ry 0 rz 160 deg; joints [0.026, 73.684, -18.298, -156.113, 57.745, 166.702]
  Set speed (17.7 mm/s)
  Call Extruder(190.24340)
  MoveL 3962 to (540.77, 452.73, 68) mm, rotated rx 180 ry 0 rz 160 deg; joints [0.198, 74.012, -18.995, -155.819, 57.447, 166.417]
  Set speed (17.7 mm/s)
  Call Extruder(197.60864)
  MoveL 3963 to (542.5, 454.28, 68) mm, rotated rx 180 ry 0 rz 160 deg; joints [0.377, 74.337, -19.685, -155.516, 57.157, 166.127]
  Set speed (17.7 mm/s)
  Call Extruder(204.87023)
  MoveL 3964 to (544.14, 455.86, 68) mm, rotated rx 180 ry 0 rz 160 deg; joints [0.559, 74.651, -20.351, -155.21, 56.881, 165.837]
  Set speed (17.7 mm/s)
  Call Extruder(208.88847)
  MoveL 3965 to (545.02, 456.76, 68) mm, rotated rx 180 ry 0 rz 160 deg; joints [0.663, 74.822, -20.713, -155.037, 56.733, 165.676]
  Set speed (17.7 mm/s)
  Call Extruder(212.88885)
  MoveL 3966 to (545.89, 457.68, 68) mm, rotated rx 180 ry 0 rz 160 deg; joints [0.767, 74.991, -21.07, -154.864, 56.589, 165.514]
  Set speed (17.7 mm/s)
  Call Extruder(217.03956)
  MoveL 3967 to (546.76, 458.64, 68) mm, rotated rx -180 ry 0 rz 160 deg; joints [0.878, 75.163, -21.433, -154.682, 56.444, 165.345]
  Call Extruder(221.00285)
  MoveL 3968 to (547.57, 459.58, 68) mm, rotated rx 180 ry 0 rz 160 deg; joints [0.985, 75.326, -21.777, -154.506, 56.308, 165.184]
  Set speed (17.7 mm/s)
  Call Extruder(225.18678)
  MoveL 3969 to (548.41, 460.59, 68) mm, rotated rx 180 ry 0 rz 160 deg; joints [1.099, 75.495, -22.134, -154.319, 56.168, 165.012]
  Set speed (17.7 mm/s)
  Call Extruder(229.20765)
  MoveL 3970 to (549.2, 461.58, 68) mm, rotated rx -180 ry 0 rz 160 deg; joints [1.211, 75.655, -22.47, -154.137, 56.039, 164.847]
  Set speed (17.7 mm/s)
  Call Extruder(233.22944)
  MoveL 3971 to (549.97, 462.58, 68) mm, rotated rx 180 ry 0 rz 160 deg; joints [1.324, 75.813, -22.803, -153.954, 55.911, 164.681]
  Set speed (17.7 mm/s)
  Call Extruder(237.30792)
  MoveL 3972 to (550.72, 463.62, 68) mm, rotated rx -180 ry 0 rz 160 deg; joints [1.441, 75.971, -23.133, -153.766, 55.787, 164.513]
  Set speed (17.7 mm/s)
  Call Extruder(241.34112)
  MoveL 3973 to (551.45, 464.65, 68) mm, rotated rx 180 ry 0 rz 160 deg; joints [1.557, 76.124, -23.454, -153.58, 55.667, 164.346]
  Call Extruder(245.42700)
  MoveL 3974 to (552.17, 465.72, 68) mm, rotated rx -180 ry 0 rz 160 deg; joints [1.676, 76.276, -23.773, -153.39, 55.551, 164.178]
  Set speed (17.7 mm/s)
  Call Extruder(249.48497)
  MoveL 3975 to (552.86, 466.79, 68) mm, rotated rx -180 ry 0 rz 160 deg; joints [1.796, 76.424, -24.083, -153.2, 55.439, 164.01]
  Set speed (17.7 mm/s)
  Call Extruder(253.60293)
  MoveL 3976 to (553.53, 467.89, 68) mm, rotated rx 180 ry 0 rz 160 deg; joints [1.919, 76.571, -24.391, -153.006, 55.329, 163.84]
  Set speed (17.7 mm/s)
  Call Extruder(257.62120)
  MoveL 3977 to (554.17, 468.98, 68) mm, rotated rx 180 ry 0 rz 160 deg; joints [2.04, 76.711, -24.685, -152.816, 55.227, 163.674]
  Set speed (17.7 mm/s)
  Call Extruder(261.74925)
  MoveL 3978 to (554.8, 470.11, 68) mm, rotated rx -180 ry 0 rz 160 deg; joints [2.166, 76.852, -24.979, -152.62, 55.126, 163.505]
  Call Extruder(265.76061)
  MoveL 3979 to (555.4, 471.22, 68) mm, rotated rx 180 ry 0 rz 160 deg; joints [2.29, 76.986, -25.258, -152.429, 55.032, 163.34]
  Set speed (17.7 mm/s)
  Call Extruder(269.85954)
  MoveL 3980 to (555.98, 472.37, 68) mm, rotated rx -180 ry 0 rz 160 deg; joints [2.417, 77.119, -25.536, -152.233, 54.941, 163.173]
  Set speed (17.7 mm/s)
  Call Extruder(275.05145)
  MoveL 3981 to (556.68, 473.84, 68) mm, rotated rx -180 ry 0 rz 160 deg; joints [2.58, 77.282, -25.876, -151.984, 54.832, 162.962]
  Set speed (17.7 mm/s)
  Call Extruder(278.04305)
  MoveL 3982 to (557.07, 474.7, 68) mm, rotated rx -180 ry 0 rz 160 deg; joints [2.675, 77.373, -26.066, -151.841, 54.773, 162.842]
  Set speed (17.7 mm/s)
  Call Extruder(286.06060)
  MoveL 3983 to (558.04, 477.02, 68) mm, rotated rx -180 ry 0 rz 160 deg; joints [2.931, 77.608, -26.554, -151.456, 54.626, 162.521]
  Set speed (17.7 mm/s)
  Call Extruder(290.25732)
  MoveL 3984 to (558.5, 478.25, 68) mm, rotated rx 180 ry 0 rz 160 deg; joints [3.067, 77.723, -26.793, -151.255, 54.558, 162.356]
  Set speed (17.7 mm/s)
